FUNCTION_BLOCK FB_Security_System_Manager
  VAR_INPUT
    VI_System_Time_MS : UDINT;
    VI_IsActivePLC : BOOL;
    VI_Arm_Request : BOOL;
    VI_Disarm_Request : BOOL;
    VI_PIN_Code : STRING(4);
    VI_RFID_Tag : STRING(20);
    VI_2FA_Code : STRING(6);
    VI_Config : ST_Security_Global_Config;
    VI_Current_TOD : TOD;
  END_VAR
  VAR_OUTPUT
    VO_Armed : BOOL;
    VO_Alarm_Active : BOOL;
    VO_Siren_Active : BOOL;
    VO_Status_Msg : STRING(200);
    VO_Send_Code_Req : BOOL;
    VO_Code_To_Send : STRING(6);
  END_VAR
  VAR_IN_OUT
    VI_Motion_Sensors : ARRAY[1..16] OF BOOL;
    VI_Door_Sensors : ARRAY[1..GVL_CONSTANTS.C_MAX_DOOR_SENSORS] OF BOOL;
    VI_Window_Sensors : ARRAY[1..16] OF BOOL;
    VI_Bypass_Motion : ARRAY[1..16] OF BOOL;
    VI_Bypass_Doors : ARRAY[1..GVL_CONSTANTS.C_MAX_DOOR_SENSORS] OF BOOL;
    VI_Bypass_Windows : ARRAY[1..16] OF BOOL;
  END_VAR
  VAR
    L_i : INT;
    L_Any_Sensor_Active : BOOL;
    L_Arm_Delay_Timer : FB_System_Timer;
    L_Alarm_Delay_Timer : FB_System_Timer;
    L_Arming_In_Progress : BOOL;
    L_Valid_PIN : BOOL;
    fbAccessCode : FB_AccessCode_Manager;
    fbTwoFactor : FB_TwoFactor_Auth;
    L_2FA_Required : BOOL;
    L_Disarm_Pending : BOOL;
    L_Reset_2FA : BOOL;
    L_Auto_Arm_Trigger : BOOL;
    R_Trig_Auto_Arm : R_TRIG;
  END_VAR

            IF NOT VI_IsActivePLC THEN
    VO_Armed := FALSE;
    VO_Alarm_Active := FALSE;
    VO_Siren_Active := FALSE;
    VO_Send_Code_Req := FALSE;
    VO_Code_To_Send := '';
    VO_Status_Msg := 'Охрана: резервный ПЛК';
    L_Arming_In_Progress := FALSE;
    L_Disarm_Pending := FALSE;
    L_2FA_Required := FALSE;
    L_Reset_2FA := FALSE;
    RETURN;
END_IF;

// 1. Проверка PIN-кода или RFID-метки через менеджер кодов
fbAccessCode(
    VI_System_Time_MS := VI_System_Time_MS,
    VI_IsActivePLC := VI_IsActivePLC,
    VI_Code_To_Check := VI_PIN_Code,
    VI_RFID_To_Check := VI_RFID_Tag,
    VI_Access_Codes := GVL_RETAIN.G_Access_Codes,
    VI_RFID_Tags := GVL_RETAIN.G_RFID_Tags,
    VO_Code_Valid => L_Valid_PIN
);

// 2. Логика постановки на охрану (с задержкой на выход)
L_Auto_Arm_Trigger := FALSE;
IF VI_Config.auto_arm_enabled THEN
    IF VI_Current_TOD >= UDINT_TO_TOD(VI_Config.auto_arm_time_ms) THEN
        L_Auto_Arm_Trigger := TRUE;
    END_IF;
END_IF;
R_Trig_Auto_Arm(CLK := L_Auto_Arm_Trigger);

IF ((VI_Arm_Request AND L_Valid_PIN) OR R_Trig_Auto_Arm.Q) AND NOT VO_Armed AND NOT L_Arming_In_Progress THEN
    // Проверка, что все двери/окна закрыты перед постановкой (с учетом байпаса)
    L_Any_Sensor_Active := FALSE;
    FOR L_i := 1 TO GVL_CONSTANTS.C_MAX_DOOR_SENSORS DO IF VI_Door_Sensors[L_i] AND NOT VI_Bypass_Doors[L_i] THEN L_Any_Sensor_Active := TRUE; END_IF; END_FOR;
    FOR L_i := 1 TO 16 DO IF VI_Window_Sensors[L_i] AND NOT VI_Bypass_Windows[L_i] THEN L_Any_Sensor_Active := TRUE; END_IF; END_FOR;
    
    IF NOT L_Any_Sensor_Active THEN
        L_Arming_In_Progress := TRUE;
        VO_Status_Msg := 'Постановка на охрану. Покиньте помещение.';
    ELSE
        VO_Status_Msg := 'Ошибка постановки: Открыты двери или окна';
    END_IF;
END_IF;

L_Arm_Delay_Timer(IN := L_Arming_In_Progress, PT := TO_TIME(VI_Config.exit_delay_seconds * 1000), VI_System_Time_MS := VI_System_Time_MS);
IF L_Arm_Delay_Timer.Q THEN
    L_Arming_In_Progress := FALSE;
    VO_Armed := TRUE;
    VO_Status_Msg := 'Система под охраной';
END_IF;

// 3. Логика снятия с охраны с 2FA
IF VI_Disarm_Request AND L_Valid_PIN AND VO_Armed THEN
    IF VI_Config.enable_2fa THEN
        L_Disarm_Pending := TRUE;
        L_2FA_Required := TRUE;
        VO_Status_Msg := 'Ожидание 2FA для снятия с охраны';
    ELSE
        // Снятие без 2FA
        VO_Armed := FALSE;
        VO_Alarm_Active := FALSE;
        VO_Siren_Active := FALSE;
        L_Arming_In_Progress := FALSE;
        VO_Status_Msg := 'Система снята с охраны';
    END_IF;
END_IF;

fbTwoFactor(
    VI_System_Time_MS := VI_System_Time_MS,
    VI_Start_Auth := L_2FA_Required,
    VI_Method := E_TwoFactor_Method.TF_METHOD_TOTP, // Для примера
    VI_User_Code := VI_2FA_Code, // Используем отдельный вход для 2FA кода
    VI_Reset_Success := L_Reset_2FA
);

VO_Send_Code_Req := fbTwoFactor.VO_Send_Code_Req;
VO_Code_To_Send := fbTwoFactor.VO_Code_To_Send;

IF L_Disarm_Pending AND fbTwoFactor.VO_State.Is_Success THEN
    VO_Armed := FALSE;
    VO_Alarm_Active := FALSE;
    VO_Siren_Active := FALSE;
    L_Arming_In_Progress := FALSE;
    L_Disarm_Pending := FALSE;
    L_2FA_Required := FALSE;
    L_Reset_2FA := TRUE;
    VO_Status_Msg := 'Система снята с охраны';
ELSIF L_Disarm_Pending AND fbTwoFactor.VO_State.Is_Locked THEN
    L_Disarm_Pending := FALSE;
    L_2FA_Required := FALSE;
    L_Reset_2FA := FALSE;
    VO_Status_Msg := 'Ошибка 2FA: Превышено количество попыток';
ELSE
    L_Reset_2FA := FALSE;
END_IF;

// 4. Логика тревоги (с задержкой на вход)
IF VO_Armed THEN
    L_Any_Sensor_Active := FALSE;
    FOR L_i := 1 TO 16 DO IF VI_Motion_Sensors[L_i] AND NOT VI_Bypass_Motion[L_i] THEN L_Any_Sensor_Active := TRUE; END_IF; END_FOR;
    FOR L_i := 1 TO GVL_CONSTANTS.C_MAX_DOOR_SENSORS DO IF VI_Door_Sensors[L_i] AND NOT VI_Bypass_Doors[L_i] THEN L_Any_Sensor_Active := TRUE; END_IF; END_FOR;
    FOR L_i := 1 TO 16 DO IF VI_Window_Sensors[L_i] AND NOT VI_Bypass_Windows[L_i] THEN L_Any_Sensor_Active := TRUE; END_IF; END_FOR;
    
    // Защелкиваем факт нарушения периметра, чтобы кратковременное срабатывание датчика не сбрасывало таймер
    IF L_Any_Sensor_Active THEN
        L_Alarm_Delay_Timer.IN := TRUE;
    END_IF;
    
    L_Alarm_Delay_Timer(PT := TO_TIME(VI_Config.entry_delay_seconds * 1000), VI_System_Time_MS := VI_System_Time_MS);
    
    IF L_Alarm_Delay_Timer.Q THEN
        VO_Alarm_Active := TRUE;
        VO_Siren_Active := TRUE;
        VO_Status_Msg := 'ТРЕВОГА! Нарушение периметра';
    ELSIF L_Alarm_Delay_Timer.IN THEN
        VO_Status_Msg := 'Внимание! Введите PIN-код для отмены тревоги';
    END_IF;
ELSE
    L_Alarm_Delay_Timer(IN := FALSE, PT := T#0s, VI_System_Time_MS := VI_System_Time_MS); // Сброс таймера при снятии с охраны
END_IF;
// >>> BULK_SYNC_ANCHOR: FB_Security_System_Manager <<<
          
END_FUNCTION_BLOCK

FUNCTION_BLOCK FB_Heating_Runtime_Diagnostics_Phase
  VAR_INPUT
    VI_Enable : BOOL;
    VI_System_Time_MS : UDINT;
  END_VAR
  VAR_OUTPUT
    VO_Executed : BOOL;
    VO_Valid : BOOL;
  END_VAR
  VAR
    fbRootCauseDiagnostics : FB_Heating_RootCause_Diagnostics;
    fbDiagEventManager : FB_Diagnostics_Event_Manager;
    L_i : INT;
    L_Any_Heating_Device_OOS : BOOL;
    L_Critical_Fault : BOOL;
    L_Device_Text : STRING(200);
    L_Critical_Text : STRING(200);
    L_Event_Text : STRING(200);
    L_Add_Text : STRING(80);
  END_VAR

            // ==============================================================================
// Heating runtime diagnostics phase
// Owns diagnostics publication for heating runtime sequencing.
// Does NOT own heating control or output decisions.
// ==============================================================================



VO_Executed := FALSE;
VO_Valid := FALSE;

IF NOT VI_Enable THEN
    RETURN;
END_IF;

// ======================================================
// ROOT CAUSE DIAGNOSTICS
// ======================================================
fbRootCauseDiagnostics(
    VI_Enable := TRUE
);

// ======================================================
// DEFAULTS
// ======================================================
L_Any_Heating_Device_OOS := FALSE;
L_Critical_Fault := FALSE;
L_Device_Text := '';
L_Critical_Text := '';
L_Event_Text := '';
L_Add_Text := '';

// ======================================================
// SERVICE / OUT-OF-SERVICE FLAGS
// ======================================================
GVL_STATUS.G_Diagnostics.Backup_Pump_Out_Of_Service :=
    NOT GVL_CONFIG.G_Backup_Circulation_Pump_In_Service;

GVL_STATUS.G_Diagnostics.Electric_Heater_Out_Of_Service :=
    NOT GVL_CONFIG.G_Electric_Heater_In_Service;

IF GVL_STATUS.G_Diagnostics.Backup_Pump_Out_Of_Service THEN
    L_Any_Heating_Device_OOS := TRUE;
    L_Add_Text := 'backup pump out of service';
    L_Device_Text := L_Add_Text;
END_IF;

IF GVL_STATUS.G_Diagnostics.Electric_Heater_Out_Of_Service THEN
    L_Any_Heating_Device_OOS := TRUE;
    L_Add_Text := 'electric heater out of service';
    IF LEN(L_Device_Text) = 0 THEN
        L_Device_Text := L_Add_Text;
    ELSIF (LEN(L_Device_Text) + LEN(L_Add_Text) + 2) < 200 THEN
        L_Device_Text := CONCAT(L_Device_Text, CONCAT('; ', L_Add_Text));
    END_IF;
END_IF;

fbDiagEventManager(
    VI_Code := GVL_CONFIG.ERR_BACKUP_PUMP_OUT_OF_SERVICE,
    VI_Severity := 2,
    VI_Active := GVL_STATUS.G_Diagnostics.Backup_Pump_Out_Of_Service,
    VI_Timestamp := VI_System_Time_MS,
    VI_Source := 400,
    VIO_Events := GVL_STATUS.G_Diagnostics_Events,
    VIO_Count := GVL_STATUS.G_Diagnostics_Count
);

fbDiagEventManager(
    VI_Code := GVL_CONFIG.ERR_ELECTRIC_HEATER_OUT_OF_SERVICE,
    VI_Severity := 2,
    VI_Active := GVL_STATUS.G_Diagnostics.Electric_Heater_Out_Of_Service,
    VI_Timestamp := VI_System_Time_MS,
    VI_Source := 401,
    VIO_Events := GVL_STATUS.G_Diagnostics_Events,
    VIO_Count := GVL_STATUS.G_Diagnostics_Count
);

FOR L_i := 1 TO GVL_CONSTANTS.C_MAX_MANIFOLDS DO

    GVL_STATUS.G_Diagnostics.Manifold_Pump_Out_Of_Service[L_i] :=
        NOT GVL_CONFIG.G_Manifold_Pump_In_Service[L_i];

    IF GVL_STATUS.G_Diagnostics.Manifold_Pump_Out_Of_Service[L_i] THEN
        L_Any_Heating_Device_OOS := TRUE;
        L_Add_Text := CONCAT('manifold pump OOS #', INT_TO_STRING(L_i));

        IF LEN(L_Device_Text) = 0 THEN
            L_Device_Text := L_Add_Text;
        ELSIF (LEN(L_Device_Text) + LEN(L_Add_Text) + 2) < 200 THEN
            L_Device_Text := CONCAT(L_Device_Text, CONCAT('; ', L_Add_Text));
        END_IF;
    END_IF;

    fbDiagEventManager(
        VI_Code := GVL_CONFIG.ERR_MANIFOLD_PUMP_OUT_OF_SERVICE,
        VI_Severity := 2,
        VI_Active := GVL_STATUS.G_Diagnostics.Manifold_Pump_Out_Of_Service[L_i],
        VI_Timestamp := VI_System_Time_MS,
        VI_Source := 410 + L_i,
        VIO_Events := GVL_STATUS.G_Diagnostics_Events,
        VIO_Count := GVL_STATUS.G_Diagnostics_Count
    );

END_FOR;

GVL_STATUS.G_Diagnostics.DHW_Heating_Pump_Out_Of_Service :=
    NOT GVL_CONFIG.G_DHW_Heating_Pump_In_Service;

GVL_STATUS.G_Diagnostics.DHW_Circ_Pump_Out_Of_Service :=
    NOT GVL_CONFIG.G_DHW_Circ_Pump_In_Service;

IF GVL_STATUS.G_Diagnostics.DHW_Heating_Pump_Out_Of_Service THEN
    L_Any_Heating_Device_OOS := TRUE;
    L_Add_Text := 'DHW heating pump out of service';

    IF LEN(L_Device_Text) = 0 THEN
        L_Device_Text := L_Add_Text;
    ELSIF (LEN(L_Device_Text) + LEN(L_Add_Text) + 2) < 200 THEN
        L_Device_Text := CONCAT(L_Device_Text, CONCAT('; ', L_Add_Text));
    END_IF;
END_IF;

IF GVL_STATUS.G_Diagnostics.DHW_Circ_Pump_Out_Of_Service THEN
    L_Any_Heating_Device_OOS := TRUE;
    L_Add_Text := 'DHW circ pump out of service';

    IF LEN(L_Device_Text) = 0 THEN
        L_Device_Text := L_Add_Text;
    ELSIF (LEN(L_Device_Text) + LEN(L_Add_Text) + 2) < 200 THEN
        L_Device_Text := CONCAT(L_Device_Text, CONCAT('; ', L_Add_Text));
    END_IF;
END_IF;

fbDiagEventManager(
    VI_Code := GVL_CONFIG.ERR_DHW_HEATING_PUMP_OUT_OF_SERVICE,
    VI_Severity := 2,
    VI_Active := GVL_STATUS.G_Diagnostics.DHW_Heating_Pump_Out_Of_Service,
    VI_Timestamp := VI_System_Time_MS,
    VI_Source := 420,
    VIO_Events := GVL_STATUS.G_Diagnostics_Events,
    VIO_Count := GVL_STATUS.G_Diagnostics_Count
);

fbDiagEventManager(
    VI_Code := GVL_CONFIG.ERR_DHW_CIRC_PUMP_OUT_OF_SERVICE,
    VI_Severity := 2,
    VI_Active := GVL_STATUS.G_Diagnostics.DHW_Circ_Pump_Out_Of_Service,
    VI_Timestamp := VI_System_Time_MS,
    VI_Source := 421,
    VIO_Events := GVL_STATUS.G_Diagnostics_Events,
    VIO_Count := GVL_STATUS.G_Diagnostics_Count
);

// ======================================================
// FREEZE HARDWARE EVENT PROJECTION
// ======================================================
L_Critical_Fault := GVL_STATE.G_Freeze_Hardware_Failed;

IF L_Critical_Fault THEN
    L_Critical_Text := 'Freeze hardware critical fault';
END_IF;

fbDiagEventManager(
    VI_Code := GVL_CONFIG.ERR_FREEZE_HARDWARE_FAILED,
    VI_Severity := 4,
    VI_Active := L_Critical_Fault,
    VI_Timestamp := VI_System_Time_MS,
    VI_Source := 430,
    VIO_Events := GVL_STATUS.G_Diagnostics_Events,
    VIO_Count := GVL_STATUS.G_Diagnostics_Count
);

GVL_STATUS.G_Diagnostics.Freeze_Hardware_Event_Pending :=
    GVL_STATUS.G_Diagnostics.Freeze_Hardware_Event_Pending OR
    L_Critical_Fault OR
    L_Any_Heating_Device_OOS;

IF L_Critical_Fault AND L_Any_Heating_Device_OOS THEN
    L_Event_Text := CONCAT(L_Critical_Text, '; ');
    IF (LEN(L_Event_Text) + LEN(L_Device_Text)) < 200 THEN
        L_Event_Text := CONCAT(L_Event_Text, L_Device_Text);
    END_IF;
    GVL_STATUS.G_Diagnostics.Freeze_Hardware_Event_Text := L_Event_Text;
ELSIF L_Critical_Fault THEN
    GVL_STATUS.G_Diagnostics.Freeze_Hardware_Event_Text := L_Critical_Text;
ELSIF L_Any_Heating_Device_OOS THEN
    GVL_STATUS.G_Diagnostics.Freeze_Hardware_Event_Text := L_Device_Text;
END_IF;

VO_Executed := TRUE;
VO_Valid := TRUE;

// >>> BULK_SYNC_ANCHOR: FB_Heating_Runtime_Diagnostics_Phase <<<
          
END_FUNCTION_BLOCK

FUNCTION_BLOCK FB_Heating_Thermal_Model
  VAR
    L_i : INT;
    L_DeltaT : REAL;
    L_Loss : REAL;
    L_Gain : REAL;
    L_Outdoor : REAL;
  END_VAR

            L_Outdoor := GVL_STATE.G_Outdoor_Temp;

FOR L_i := 1 TO GVL_CONSTANTS.C_MAX_ZONES DO

    L_DeltaT := GVL_STATE.G_Room_Temps[L_i] - L_Outdoor;

    L_Loss := L_DeltaT * REAL#0.01 * GVL_HEATING_POLICY.G_Zone_Thermal_Inertia[L_i];

    L_Gain := (GVL_STATE.G_Floor_Temps[L_i] - GVL_STATE.G_Room_Temps[L_i]) * REAL#0.05;

    GVL_HEATING_POLICY.G_Zone_Heat_Loss_Rate[L_i] := L_Loss;
    GVL_HEATING_POLICY.G_Zone_Heat_Gain_Rate[L_i] := L_Gain;

    GVL_HEATING_POLICY.G_Zone_Thermal_Response[L_i] := L_Gain - L_Loss;

    GVL_HEATING_POLICY.G_Zone_Thermal_Demand[L_i] := 
        GVL_STATE.G_Target_Temperature - GVL_STATE.G_Room_Temps[L_i];

    IF ABS(GVL_HEATING_POLICY.G_Zone_Thermal_Response[L_i]) > REAL#0.01 THEN
        GVL_HEATING_POLICY.G_Zone_Time_To_Heat_MS[L_i] := 
            REAL_TO_UDINT(ABS(GVL_HEATING_POLICY.G_Zone_Thermal_Demand[L_i] /
                  GVL_HEATING_POLICY.G_Zone_Thermal_Response[L_i]) * REAL#60000.0);
    ELSE
        GVL_HEATING_POLICY.G_Zone_Time_To_Heat_MS[L_i] := 0;
    END_IF;

    GVL_HEATING_POLICY.G_Zone_Predicted_Temp_30m[L_i] :=
        GVL_STATE.G_Room_Temps[L_i] + 
        GVL_HEATING_POLICY.G_Zone_Thermal_Response[L_i] * REAL#30.0;

    GVL_HEATING_POLICY.G_Zone_Thermal_Model_Confidence[L_i] :=
        LIMIT(REAL#0.0, REAL#1.0, ABS(GVL_HEATING_POLICY.G_Zone_Thermal_Response[L_i]));

END_FOR;
          
END_FUNCTION_BLOCK

FUNCTION_BLOCK FB_Gateway_Interface
  VAR_INPUT
    VI_System_Time_MS : UDINT;
    VI_Local_PLC_Role : E_PLC_ROLE;
    VI_Incoming_Command : ST_Gateway_Command;
    VI_Command_Received : BOOL;
    VI_Outdoor_Temp : REAL;
    VI_Security_Armed : BOOL;
    VI_Flood_Alarm_Active : BOOL;
    VI_Gas_Alarm_Active : BOOL;
    VI_Fire_Alarm_Active : BOOL;
    VI_Methane_Concentration : REAL;
    VI_Active_Scenario : E_SCENARIO_TYPE;
    VI_Send_2FA_Req : BOOL;
    VI_2FA_Code : STRING(6);
  END_VAR
  VAR_OUTPUT
    VO_Modbus_Registers : ARRAY[0..GVL_CONSTANTS.C_MAX_MODBUS_REGISTERS-1] OF WORD;
    VO_Lighting_Override : ARRAY[1..GVL_CONSTANTS.C_MAX_LIGHT_ZONES] OF BYTE;
    VO_Blinds_Override : ARRAY[1..GVL_CONSTANTS.C_MAX_BLINDS] OF BYTE;
    VO_Socket_Override : ARRAY[1..GVL_CONSTANTS.C_MAX_SOCKETS] OF BOOL;
    VO_Arm_Req : BOOL;
    VO_Disarm_Req : BOOL;
    VO_PIN_Code : STRING(4);
    VO_RFID_Tag : STRING(20);
    VO_2FA_Code_In : STRING(6);
    VO_Data_Ready : BOOL;
    VO_HMI_Status_Message : STRING(200);
    VO_Telegram_Msg : STRING(200);
    VO_Send_Telegram : BOOL;
    VO_Set_Scenario_Req : BOOL;
    VO_Target_Scenario : E_SCENARIO_TYPE;
    VO_Set_Temp_Req : BOOL;
    VO_Target_Zone : INT;
    VO_Target_Temp : REAL;
    VO_Set_Vent_Req : BOOL;
    VO_Target_Vent_Speed : BYTE;
    VO_Reset_Errors_Req : BOOL;
    VO_Set_Config_Req : BOOL;
    VO_Sync_Time_Req : BOOL;
    VO_New_Time_MS : UDINT;
  END_VAR
  VAR_IN_OUT
    VI_FloorHeating_Temps : ARRAY[1..GVL_CONSTANTS.C_MAX_HEATING_CIRCUITS] OF REAL;
    VI_Room_Temps : ARRAY[1..GVL_CONSTANTS.C_MAX_ZONES] OF REAL;
    VI_Zone_Valve_States : ARRAY[1..GVL_CONSTANTS.C_MAX_HEATING_CIRCUITS] OF BOOL;
    VI_Manifold_Pressures : ARRAY[1..GVL_CONSTANTS.C_MAX_MANIFOLDS] OF REAL;
    VI_Manifold_Pump_States : ARRAY[1..GVL_CONSTANTS.C_MAX_MANIFOLDS] OF BOOL;
    VI_Lighting_Base_Levels : ARRAY[1..GVL_CONSTANTS.C_MAX_LIGHT_ZONES] OF BYTE;
    VI_Socket_States : ARRAY[1..GVL_CONSTANTS.C_MAX_SOCKETS] OF BOOL;
    VI_Blinds_Positions : ARRAY[1..GVL_CONSTANTS.C_MAX_BLINDS] OF BYTE;
    VI_Allowed_IPs : ARRAY[1..GVL_CONSTANTS.C_MAX_ALLOWED_IPS] OF STRING(15);
  END_VAR
  VAR
    L_last_update_time : UDINT;
    L_i : INT;
    L_j : INT;
    L_idx : INT;
    L_tmp_word : WORD;
    L_Code_UDINT : UDINT;
    L_Prev_Fire : BOOL;
    L_Prev_Gas : BOOL;
    L_Prev_Flood : BOOL;
    L_Prev_Security : BOOL;
    L_Deduplicator : FB_Command_Deduplication;
    L_CRC_Calc : FB_CRC32_Calculator;
    L_Calculated_CRC : DWORD;
    L_IP_Allowed : BOOL;
    L_Process_Command : ST_Gateway_Command;
    L_Has_Command_To_Process : BOOL;
  END_VAR
  VAR RETAIN
    L_Command_Buffer : ARRAY[1..GVL_CONSTANTS.C_MAX_GATEWAY_COMMANDS] OF ST_Gateway_Command;
    L_Buffer_Head : INT := 1;
    L_Buffer_Tail : INT := 1;
    L_Buffer_Count : INT := 0;
  END_VAR

            VO_Send_Telegram := FALSE;
IF VI_Fire_Alarm_Active AND NOT L_Prev_Fire THEN
    VO_Telegram_Msg := 'ВНИМАНИЕ! ПОЖАРНАЯ ТРЕВОГА!';
    VO_Send_Telegram := TRUE;
END_IF;
IF VI_Gas_Alarm_Active AND NOT L_Prev_Gas THEN
    VO_Telegram_Msg := 'ВНИМАНИЕ! УТЕЧКА ГАЗА!';
    VO_Send_Telegram := TRUE;
END_IF;
IF VI_Flood_Alarm_Active AND NOT L_Prev_Flood THEN
    VO_Telegram_Msg := 'ВНИМАНИЕ! ПРОТЕЧКА ВОДЫ!';
    VO_Send_Telegram := TRUE;
END_IF;
IF VI_Security_Armed AND NOT L_Prev_Security THEN
    VO_Telegram_Msg := 'ОХРАНА ВКЛЮЧЕНА';
    VO_Send_Telegram := TRUE;
ELSIF NOT VI_Security_Armed AND L_Prev_Security THEN
    VO_Telegram_Msg := 'ОХРАНА ОТКЛЮЧЕНА';
    VO_Send_Telegram := TRUE;
END_IF;

L_Prev_Fire := VI_Fire_Alarm_Active;
L_Prev_Gas := VI_Gas_Alarm_Active;
L_Prev_Flood := VI_Flood_Alarm_Active;
L_Prev_Security := VI_Security_Armed;

IF (VI_System_Time_MS - L_last_update_time) >= GVL_CONSTANTS.C_MS_IN_SECOND THEN
    L_last_update_time := VI_System_Time_MS;
    L_tmp_word := 0;
    IF VI_Local_PLC_Role = E_PLC_ROLE.ROLE_ACTIVE THEN L_tmp_word := L_tmp_word OR 1; END_IF;
    IF VI_Security_Armed THEN L_tmp_word := L_tmp_word OR 2; END_IF;
    IF VI_Flood_Alarm_Active THEN L_tmp_word := L_tmp_word OR 4; END_IF;
    IF VI_Gas_Alarm_Active THEN L_tmp_word := L_tmp_word OR 8; END_IF;
    IF VI_Fire_Alarm_Active THEN L_tmp_word := L_tmp_word OR 16; END_IF;
    VO_Modbus_Registers[0] := L_tmp_word;

    FOR L_i := 1 TO GVL_CONSTANTS.C_MAX_HEATING_CIRCUITS DO
        VO_Modbus_Registers[L_i] := TO_WORD(TO_INT(VI_FloorHeating_Temps[L_i] * REAL#10.0));
    END_FOR;

    FOR L_i := 1 TO GVL_CONSTANTS.C_MAX_ZONES DO
        VO_Modbus_Registers[16 + L_i] := TO_WORD(TO_INT(VI_Room_Temps[L_i] * REAL#10.0));
    END_FOR;

    L_tmp_word := 0;
    FOR L_i := 1 TO GVL_CONSTANTS.C_MAX_HEATING_CIRCUITS DO
        IF VI_Zone_Valve_States[L_i] THEN
            L_tmp_word := L_tmp_word OR SHL(TO_WORD(1), L_i - 1);
        END_IF;
    END_FOR;
    VO_Modbus_Registers[33] := L_tmp_word;

    FOR L_i := 1 TO GVL_CONSTANTS.C_MAX_MANIFOLDS DO
        VO_Modbus_Registers[33 + L_i] := TO_WORD(TO_INT(VI_Manifold_Pressures[L_i] * REAL#100.0));
    END_FOR;

    FOR L_i := 1 TO GVL_CONSTANTS.C_MAX_LIGHT_ZONES DO
        VO_Modbus_Registers[39 + L_i] := TO_WORD(VI_Lighting_Base_Levels[L_i]);
    END_FOR;

    FOR L_i := 1 TO GVL_CONSTANTS.C_MAX_BLINDS DO
        VO_Modbus_Registers[71 + L_i] := TO_WORD(VI_Blinds_Positions[L_i]);
    END_FOR;

    FOR L_i := 0 TO (GVL_CONSTANTS.C_MAX_SOCKETS - 1) / 16 DO
        L_tmp_word := 0;
        FOR L_j := 1 TO 16 DO
            L_idx := (L_i * 16) + L_j;
            IF L_idx <= GVL_CONSTANTS.C_MAX_SOCKETS THEN
                IF VI_Socket_States[L_idx] THEN
                    L_tmp_word := L_tmp_word OR SHL(TO_WORD(1), L_j - 1);
                END_IF;
            END_IF;
        END_FOR;
        VO_Modbus_Registers[92 + L_i] := L_tmp_word;
    END_FOR;

    VO_Modbus_Registers[100] := SEL(VI_Send_2FA_Req, 0, 1);
    IF VI_Send_2FA_Req THEN
        L_Code_UDINT := STRING_TO_UDINT(VI_2FA_Code);
        VO_Modbus_Registers[101] := TO_WORD(L_Code_UDINT AND 16#FFFF);
        VO_Modbus_Registers[102] := TO_WORD(SHR(L_Code_UDINT, 16));
    ELSE
        VO_Modbus_Registers[101] := 0;
        VO_Modbus_Registers[102] := 0;
    END_IF;

    VO_Data_Ready := TRUE;
END_IF;

VO_Arm_Req := FALSE;
VO_Disarm_Req := FALSE;
VO_Set_Scenario_Req := FALSE;
VO_Set_Temp_Req := FALSE;
VO_Set_Vent_Req := FALSE;
VO_Reset_Errors_Req := FALSE;
VO_Set_Config_Req := FALSE;
VO_Sync_Time_Req := FALSE;
L_Has_Command_To_Process := FALSE;

IF VI_Command_Received THEN
    IF VI_Local_PLC_Role = E_PLC_ROLE.ROLE_ACTIVE THEN
        L_Process_Command := VI_Incoming_Command;
        L_Has_Command_To_Process := TRUE;
    ELSE
        IF L_Buffer_Count < GVL_CONSTANTS.C_MAX_GATEWAY_COMMANDS THEN
            L_Command_Buffer[L_Buffer_Head] := VI_Incoming_Command;
            L_Buffer_Head := L_Buffer_Head + 1;
            IF L_Buffer_Head > GVL_CONSTANTS.C_MAX_GATEWAY_COMMANDS THEN L_Buffer_Head := 1; END_IF;
            L_Buffer_Count := L_Buffer_Count + 1;
        END_IF;
    END_IF;
END_IF;

IF NOT L_Has_Command_To_Process AND (VI_Local_PLC_Role = E_PLC_ROLE.ROLE_ACTIVE) AND (L_Buffer_Count > 0) THEN
    L_Process_Command := L_Command_Buffer[L_Buffer_Tail];
    L_Buffer_Tail := L_Buffer_Tail + 1;
    IF L_Buffer_Tail > GVL_CONSTANTS.C_MAX_GATEWAY_COMMANDS THEN L_Buffer_Tail := 1; END_IF;
    L_Buffer_Count := L_Buffer_Count - 1;
    L_Has_Command_To_Process := TRUE;
END_IF;

IF L_Has_Command_To_Process THEN
    L_IP_Allowed := FALSE;
    IF L_Process_Command.source_ip = '' THEN
        L_IP_Allowed := TRUE;
    ELSE
        FOR L_i := 1 TO GVL_CONSTANTS.C_MAX_ALLOWED_IPS DO
            IF VI_Allowed_IPs[L_i] = L_Process_Command.source_ip THEN
                L_IP_Allowed := TRUE;
                EXIT;
            END_IF;
        END_FOR;
    END_IF;

    IF NOT L_IP_Allowed THEN
        VO_HMI_Status_Message := 'Gateway: Ошибка безопасности (Неизвестный IP)';
        RETURN;
    END_IF;

    L_CRC_Calc();
    L_Calculated_CRC := L_CRC_Calc.VO_CRC;

    IF L_Calculated_CRC = L_Process_Command.crc32 THEN
        L_Deduplicator(VI_Command_ID := L_Process_Command.command_id, VI_Command_Type := L_Process_Command.command_type, VI_Command_Value := L_Process_Command.target_value, VI_System_Time_MS := VI_System_Time_MS);

        IF L_Deduplicator.VO_Is_New_Command THEN
            CASE L_Process_Command.command_type OF
                E_Gateway_Command_Type.CMD_SET_SCENARIO:
                    VO_Set_Scenario_Req := TRUE;
                    VO_Target_Scenario := L_Process_Command.target_scenario;
                    VO_HMI_Status_Message := 'Gateway: Сценарий изменен';
                E_Gateway_Command_Type.CMD_SET_LIGHT:
                    IF (L_Process_Command.target_zone >= 1) AND (L_Process_Command.target_zone <= GVL_CONSTANTS.C_MAX_LIGHT_ZONES) THEN
                        VO_Lighting_Override[L_Process_Command.target_zone] := TO_BYTE(L_Process_Command.target_value);
                        VO_HMI_Status_Message := 'Gateway: Команда освещения принята';
                    END_IF;
                E_Gateway_Command_Type.CMD_SET_BLINDS:
                    IF (L_Process_Command.target_zone >= 1) AND (L_Process_Command.target_zone <= GVL_CONSTANTS.C_MAX_BLINDS) THEN
                        VO_Blinds_Override[L_Process_Command.target_zone] := TO_BYTE(L_Process_Command.target_value);
                        VO_HMI_Status_Message := 'Gateway: Команда штор принята';
                    END_IF;
                E_Gateway_Command_Type.CMD_SET_SOCKET:
                    IF (L_Process_Command.target_zone >= 1) AND (L_Process_Command.target_zone <= GVL_CONSTANTS.C_MAX_SOCKETS) THEN
                        VO_Socket_Override[L_Process_Command.target_zone] := L_Process_Command.target_on_off;
                        VO_HMI_Status_Message := 'Gateway: Команда розетки принята';
                    END_IF;
                E_Gateway_Command_Type.CMD_SET_SECURITY:
                    IF L_Process_Command.target_armed THEN VO_Arm_Req := TRUE; ELSE VO_Disarm_Req := TRUE; END_IF;
                    VO_PIN_Code := L_Process_Command.target_pin;
                    VO_2FA_Code_In := L_Process_Command.target_2fa_code;
                    VO_HMI_Status_Message := 'Gateway: Запрос охраны принят';
                E_Gateway_Command_Type.CMD_SET_TEMP:
                    IF (L_Process_Command.target_zone >= 1) AND (L_Process_Command.target_zone <= GVL_CONSTANTS.C_MAX_HEATING_CIRCUITS) THEN
                        VO_Set_Temp_Req := TRUE;
                        VO_Target_Zone := L_Process_Command.target_zone;
                        VO_Target_Temp := L_Process_Command.target_value;
                        VO_HMI_Status_Message := 'Gateway: Уставка температуры изменена';
                    END_IF;
                E_Gateway_Command_Type.CMD_SET_VENT:
                    VO_Set_Vent_Req := TRUE;
                    VO_Target_Vent_Speed := TO_BYTE(L_Process_Command.target_value);
                    VO_HMI_Status_Message := 'Gateway: Уставка вентиляции изменена';
                E_Gateway_Command_Type.CMD_TELEGRAM_MSG:
                    VO_Telegram_Msg := L_Process_Command.telegram_msg;
                    VO_Send_Telegram := TRUE;
                    VO_HMI_Status_Message := 'Gateway: Сообщение Telegram отправлено';
                E_Gateway_Command_Type.CMD_SYNC_TIME:
                    VO_Sync_Time_Req := TRUE;
                    VO_New_Time_MS := REAL_TO_UDINT(L_Process_Command.target_value);
                    VO_HMI_Status_Message := 'Gateway: Время синхронизировано';
                E_Gateway_Command_Type.CMD_RESET_ERRORS:
                    VO_Reset_Errors_Req := TRUE;
                    VO_HMI_Status_Message := 'Gateway: Запрос на сброс ошибок принят';
                E_Gateway_Command_Type.CMD_SET_CONFIG:
                    VO_Set_Config_Req := TRUE;
                    VO_HMI_Status_Message := 'Gateway: Запрос на применение конфигурации принят';
            END_CASE;
        END_IF;
    ELSE
        VO_HMI_Status_Message := 'Gateway: Ошибка CRC команды';
    END_IF;
END_IF;

// >>> BULK_SYNC_ANCHOR: FB_Gateway_Interface <<<
          
END_FUNCTION_BLOCK

FUNCTION_BLOCK FB_Heating_Manifold_Control
  VAR_INPUT
    VI_System_Time_MS : UDINT;
    VI_IsActivePLC : BOOL;
    VI_DHW_Heating_Demand : BOOL;
    VI_Freeze_Mode_Active : BOOL;
    VI_Target_Supply_Temp : REAL;
    VI_Any_Zone_Active : ARRAY[1..GVL_CONSTANTS.C_MAX_MANIFOLDS] OF BOOL;
  END_VAR
  VAR_OUTPUT
    VO_Manifold_Pumps : ARRAY[1..GVL_CONSTANTS.C_MAX_MANIFOLDS] OF BOOL;
    VO_Manifold_Valves : ARRAY[1..GVL_CONSTANTS.C_MAX_MANIFOLDS] OF REAL;
    VO_Status : ARRAY[1..GVL_CONSTANTS.C_MAX_MANIFOLDS] OF ST_Manifold_Status;
  END_VAR
  VAR_IN_OUT
    VI_Manifold_Pressures : ARRAY[1..GVL_CONSTANTS.C_MAX_MANIFOLDS] OF REAL;
    VI_Manifold_Currents : ARRAY[1..GVL_CONSTANTS.C_MAX_MANIFOLDS] OF REAL;
    VI_Manifold_Temps_Supply : ARRAY[1..GVL_CONSTANTS.C_MAX_MANIFOLDS] OF REAL;
    VI_Manifold_Temps_Return : ARRAY[1..GVL_CONSTANTS.C_MAX_MANIFOLDS] OF REAL;
  END_VAR
  VAR
    L_i : INT;
    L_Delta_T : REAL;
    L_PID_Valves : ARRAY[1..GVL_CONSTANTS.C_MAX_MANIFOLDS] OF FB_PID_Controller;
    L_PID_Timer : ARRAY[1..GVL_CONSTANTS.C_MAX_MANIFOLDS] OF FB_System_Timer;
    L_Pump_Run_Timer : ARRAY[1..GVL_CONSTANTS.C_MAX_MANIFOLDS] OF FB_System_Timer;
    L_Pump_Pause_Timer : ARRAY[1..GVL_CONSTANTS.C_MAX_MANIFOLDS] OF FB_System_Timer;
    L_Pump_In_Pause : ARRAY[1..GVL_CONSTANTS.C_MAX_MANIFOLDS] OF BOOL;
    L_Pump_Diag : ARRAY[1..GVL_CONSTANTS.C_MAX_MANIFOLDS] OF FB_Device_Predictive_Diag;
  END_VAR

            // ==============================================================================
// Heating manifold control helper
// Internal refactoring helper for FB_Heating_System_Manager.
// Valve test override remains in FB_Heating_System_Manager for now.
// ==============================================================================



FOR L_i := 1 TO GVL_CONSTANTS.C_MAX_MANIFOLDS DO
    L_PID_Timer[L_i](IN := TRUE, PT := T#1s, VI_System_Time_MS := VI_System_Time_MS);
    IF L_PID_Timer[L_i].Q THEN
        L_PID_Timer[L_i](IN := FALSE, PT := T#1s, VI_System_Time_MS := VI_System_Time_MS);
        L_PID_Timer[L_i](IN := TRUE, PT := T#1s, VI_System_Time_MS := VI_System_Time_MS);

        L_PID_Valves[L_i](
            VI_SetPoint := VI_Target_Supply_Temp,
            VI_ProcessValue := VI_Manifold_Temps_Supply[L_i],
            VI_Kp := 2.0,
            VI_Tn := 120.0,
            VI_Tv := 0.0,
            VI_Y_Min := 0.0,
            VI_Y_Max := 100.0,
            VI_Cycle_Time_S := 1.0,
            VO_Output => VO_Manifold_Valves[L_i]
        );
    END_IF;

    L_Pump_Run_Timer[L_i](
        IN := VO_Manifold_Pumps[L_i] AND NOT L_Pump_In_Pause[L_i],
        PT := T#72h,
        VI_System_Time_MS := VI_System_Time_MS
    );
    IF L_Pump_Run_Timer[L_i].Q THEN
        L_Pump_In_Pause[L_i] := TRUE;
    END_IF;

    L_Pump_Pause_Timer[L_i](
        IN := L_Pump_In_Pause[L_i],
        PT := T#1h,
        VI_System_Time_MS := VI_System_Time_MS
    );
    IF L_Pump_Pause_Timer[L_i].Q THEN
        L_Pump_In_Pause[L_i] := FALSE;
    END_IF;

    IF VI_DHW_Heating_Demand THEN
        VO_Manifold_Pumps[L_i] := FALSE;
        VO_Manifold_Valves[L_i] := 0.0;
    ELSE
        VO_Manifold_Pumps[L_i] := VI_IsActivePLC AND VI_Any_Zone_Active[L_i] AND NOT L_Pump_In_Pause[L_i];
    END_IF;

    IF VI_Freeze_Mode_Active THEN
        VO_Manifold_Pumps[L_i] := TRUE;
        IF VO_Manifold_Valves[L_i] < 35.0 THEN
            VO_Manifold_Valves[L_i] := 35.0;
        END_IF;
    END_IF;

    VO_Status[L_i].Pump_On := VO_Manifold_Pumps[L_i];
    VO_Status[L_i].Pump_Current := VI_Manifold_Currents[L_i];
    VO_Status[L_i].Pressure := VI_Manifold_Pressures[L_i];
    VO_Status[L_i].Temp_Supply := VI_Manifold_Temps_Supply[L_i];
    VO_Status[L_i].Temp_Return := VI_Manifold_Temps_Return[L_i];
    VO_Status[L_i].Valve_Pos := VO_Manifold_Valves[L_i];

    L_Pump_Diag[L_i](
        VI_Current_Value := VI_Manifold_Currents[L_i],
        VI_Nominal_Value := 0.55,
        VI_Is_Running := VO_Manifold_Pumps[L_i],
        VI_Reset_Stats := FALSE,
        VI_System_Time_MS := VI_System_Time_MS,
        VIO_Health_Data := VO_Status[L_i].Health
    );

    IF VO_Manifold_Pumps[L_i] THEN
        L_Delta_T := VI_Manifold_Temps_Supply[L_i] - VI_Manifold_Temps_Return[L_i];

        VO_Status[L_i].Error := FALSE;
        VO_Status[L_i].Error_ID := 0;

        IF VI_Manifold_Currents[L_i] <= 0.01 THEN
            VO_Status[L_i].Error := TRUE;
            VO_Status[L_i].Error_ID := TO_WORD(GVL_CONFIG.ERR_PUMP_NO_CURRENT);
        ELSIF VI_Manifold_Currents[L_i] < 0.3 THEN
            VO_Status[L_i].Error := TRUE;
            VO_Status[L_i].Error_ID := TO_WORD(GVL_CONFIG.ERR_PUMP_UNDERCURRENT);
        ELSIF VI_Manifold_Currents[L_i] > 1.5 THEN
            VO_Status[L_i].Error := TRUE;
            VO_Status[L_i].Error_ID := TO_WORD(GVL_CONFIG.ERR_PUMP_OVERCURRENT);
        END_IF;

        IF (NOT VO_Status[L_i].Error) AND ((VI_Manifold_Pressures[L_i] < 1.5) OR (VI_Manifold_Pressures[L_i] > 2.5)) THEN
            VO_Status[L_i].Error := TRUE;
            VO_Status[L_i].Error_ID := TO_WORD(GVL_CONFIG.ERR_PRESSURE_OUT_OF_RANGE);
        END_IF;

        IF NOT VO_Status[L_i].Error THEN
            IF L_Delta_T < 5.0 THEN
                VO_Status[L_i].Error := TRUE;
                VO_Status[L_i].Error_ID := TO_WORD(GVL_CONFIG.ERR_DELTA_T_LOW);
            ELSIF L_Delta_T > 10.0 THEN
                VO_Status[L_i].Error := TRUE;
                VO_Status[L_i].Error_ID := TO_WORD(GVL_CONFIG.ERR_DELTA_T_HIGH);
            END_IF;
        END_IF;
    END_IF;
END_FOR;

// >>> BULK_SYNC_ANCHOR: FB_Heating_Manifold_Control <<<
          
END_FUNCTION_BLOCK

FUNCTION_BLOCK FB_Distributed_Orchestration_Runtime
  VAR_INPUT
    VI_Enable : BOOL;
    VI_System_Time_MS : UDINT;
  END_VAR
  VAR
    L_State : ST_Distributed_Orchestration_State;
    L_Finalized_Runtime_Continuity : BOOL;
  END_VAR

            IF NOT VI_Enable THEN
    GVL_Distributed_Orchestration.G_Runtime_Valid := FALSE;
    RETURN;
END_IF;

L_State.Runtime_Valid := TRUE;
L_State.Runtime_System_Time_MS := VI_System_Time_MS;

L_State.Orchestration_Sequence_Id :=
    GVL_Distributed_Orchestration.G_Last_Distributed_Sequence_Id + 1;

L_State.Distributed_Execution_Active := TRUE;

L_State.Cross_Node_Isolation_Required :=
    GVL_Distributed_Orchestration.G_Cross_Node_Isolation_Active;

L_State.Cross_Node_Recovery_Required :=
    GVL_Distributed_Orchestration.G_Cross_Node_Recovery_Active;

L_State.Cross_Node_Rollback_Required :=
    GVL_Distributed_Orchestration.G_Cross_Node_Rollback_Active;

L_Finalized_Runtime_Continuity :=
    GVL_SEMANTIC_PROGRESS.Semantic_Forward_Progress_Valid
    AND GVL_SEMANTIC_PROGRESS.Semantic_Execution_Continuity_OK
    AND NOT GVL_SEMANTIC_PROGRESS.Semantic_Progress_Lease_Expired
    AND NOT GVL_SEMANTIC_PROGRESS.Semantic_Progress_Quarantine_Active
    AND GVL_RUNTIME_SNAPSHOT.Snapshot_Frozen
    AND GVL_RUNTIME_SNAPSHOT.Snapshot_Publication_Allowed
    AND GVL_RUNTIME_SNAPSHOT.Snapshot_Copy_Valid
    AND GVL_RUNTIME_SNAPSHOT.Snapshot_Isolation_Valid
    AND NOT GVL_RUNTIME_SNAPSHOT.Snapshot_Mutation_Detected
    AND GVL_DISTRIBUTED_SNAPSHOT.Distributed_Publication_Reconciled
    AND GVL_DISTRIBUTED_SNAPSHOT.Distributed_Publication_Freeze_Valid
    AND GVL_DISTRIBUTED_SNAPSHOT.Distributed_Snapshot_Consistent
    AND GVL_DISTRIBUTED_COMMIT.Distributed_Commit_Valid
    AND GVL_DISTRIBUTED_COMMIT.Publication_Prepare_Valid
    AND GVL_DISTRIBUTED_COMMIT.Publication_Commit_Confirmed
    AND NOT GVL_DISTRIBUTED_COMMIT.Peer_Commit_Mismatch
    AND NOT GVL_DISTRIBUTED_COMMIT.Commit_Lease_Expired
    AND GVL_OUTPUT_EPOCH.Output_Publication_Valid
    AND GVL_OUTPUT_EPOCH.Output_Runtime_Epoch_Valid
    AND NOT GVL_OUTPUT_EPOCH.Output_Lease_Expired
    AND NOT GVL_OUTPUT_EPOCH.Output_Forced_Safe_Decay
    AND GVL_COMMAND_VERIFY.PreOutput_Barrier_OK
    AND NOT GVL_COMMAND_VERIFY.PreOutput_Block_IO;

L_State.Distributed_Scheduler_Healthy :=
    GVL_Runtime_Bus.G_TX_Healthy
    AND GVL_Distributed_Runtime.G_Distributed_Authority_Healthy
    AND L_Finalized_Runtime_Continuity;

L_State.Distributed_Timing_Window_Valid :=
    GVL_Distributed_Authority.G_Distributed_Safety_Barrier_OK
    AND L_Finalized_Runtime_Continuity;

IF L_State.Distributed_Scheduler_Healthy
   AND L_State.Distributed_Timing_Window_Valid THEN
    L_State.Distributed_Projection_Granted := TRUE;
    L_State.Distributed_Recovery_Allowed := TRUE;
    L_State.Distributed_Rollback_Allowed := TRUE;
    L_State.Status_Code := 0;
    L_State.Status_Text := 'Distributed orchestration runtime healthy';
ELSE
    L_State.Distributed_Projection_Blocked := TRUE;
    L_State.Distributed_Conflict_Detected := TRUE;
    L_State.Status_Code := 2;
    L_State.Status_Text := 'Distributed orchestration blocked';
END_IF;

IF GVL_Distributed_Runtime.G_Split_Brain_Suspected THEN
    L_State.Distributed_Split_Execution_Suspected := TRUE;
    L_State.Distributed_Projection_Blocked := TRUE;
    L_State.Status_Code := 3;
    L_State.Status_Text := 'Distributed split execution suspected';
END_IF;

GVL_Distributed_Orchestration.G_Orchestration_State := L_State;
GVL_Distributed_Orchestration.G_Last_Distributed_Sequence_Id := L_State.Orchestration_Sequence_Id;
GVL_Distributed_Orchestration.G_Distributed_Projection_Healthy := L_State.Distributed_Projection_Granted;
GVL_Distributed_Orchestration.G_Distributed_Scheduler_Healthy := L_State.Distributed_Scheduler_Healthy;
GVL_Distributed_Orchestration.G_Runtime_Valid := TRUE;
GVL_Distributed_Orchestration.G_Last_Update_MS := VI_System_Time_MS;
GVL_Distributed_Orchestration.G_Status_Code := L_State.Status_Code;
GVL_Distributed_Orchestration.G_Status_Text := L_State.Status_Text;
          
END_FUNCTION_BLOCK

FUNCTION_BLOCK FB_Boiler_Cascade_Manager
  VAR_INPUT
    VI_Enable : BOOL;
    VI_System_Time_MS : UDINT;
    VI_Boiler_Stop : BOOL;
    VI_DHW_Heating_Demand : BOOL;
    VI_DHW_Target_Temp : REAL;
    VI_Target_Supply_Temp : REAL;
    VI_Demand_Power : REAL;
    VI_Boiler_Flame_Status : ARRAY[1..GVL_CONSTANTS.C_MAX_BOILERS] OF BOOL;
    VI_Boiler_Error_Status : ARRAY[1..GVL_CONSTANTS.C_MAX_BOILERS] OF BOOL;
    VI_Boiler_OT_Online : ARRAY[1..GVL_CONSTANTS.C_MAX_BOILERS] OF BOOL;
    VI_Boiler_Modulation : ARRAY[1..GVL_CONSTANTS.C_MAX_BOILERS] OF REAL;
  END_VAR
  VAR_OUTPUT
    VO_Boiler_Enable : ARRAY[1..GVL_CONSTANTS.C_MAX_BOILERS] OF BOOL;
    VO_Boiler_Setpoint : ARRAY[1..GVL_CONSTANTS.C_MAX_BOILERS] OF REAL;
    VO_Lead_Boiler : BYTE;
  END_VAR
  VAR
    L_i : INT;
    L_Lead_Boiler : BYTE := 1;
    L_Last_Rotation_MS : UDINT := 0;
    L_Rotation_Initialized : BOOL := FALSE;
    L_Rotation_Period_MS : UDINT := 604800000;
    L_Lead_Available : BOOL;
    L_Reserve_Available : BOOL;
    L_Reserve_Boiler : BYTE;
    L_Start_Reserve : BOOL;
    L_Target_Setpoint : REAL;
    L_Flame_Miss_Timer : ARRAY[1..GVL_CONSTANTS.C_MAX_BOILERS] OF TON;
  END_VAR

            // Сброс выходов по умолчанию
FOR L_i := 1 TO GVL_CONSTANTS.C_MAX_BOILERS DO
    VO_Boiler_Enable[L_i] := FALSE;
    VO_Boiler_Setpoint[L_i] := 0.0;
END_FOR;

// Инициализация ротации
IF NOT L_Rotation_Initialized THEN
    L_Last_Rotation_MS := VI_System_Time_MS;
    L_Rotation_Initialized := TRUE;
END_IF;

// Принудительная остановка
IF VI_Boiler_Stop THEN
    VO_Lead_Boiler := L_Lead_Boiler;
    RETURN;
END_IF;

// Ротация строго каждые 168 часов
IF (VI_System_Time_MS - L_Last_Rotation_MS) >= L_Rotation_Period_MS THEN
    IF GVL_CONSTANTS.C_MAX_BOILERS > 1 THEN
        L_Lead_Boiler := 3 - L_Lead_Boiler;
    END_IF;
    L_Last_Rotation_MS := VI_System_Time_MS;
END_IF;

L_Reserve_Boiler := SEL(L_Lead_Boiler = 1, 1, 2);

L_Lead_Available :=
    VI_Boiler_OT_Online[L_Lead_Boiler] AND
    NOT VI_Boiler_Error_Status[L_Lead_Boiler];

L_Reserve_Available :=
    (GVL_CONSTANTS.C_MAX_BOILERS > 1) AND
    VI_Boiler_OT_Online[L_Reserve_Boiler] AND
    NOT VI_Boiler_Error_Status[L_Reserve_Boiler];

// Контроль "команда есть, пламени нет" для ведущего котла
L_Flame_Miss_Timer[L_Lead_Boiler](
    IN := VI_Enable AND L_Lead_Available AND NOT VI_DHW_Heating_Demand AND NOT VI_Boiler_Flame_Status[L_Lead_Boiler],
    PT := T#120s
);

IF L_Flame_Miss_Timer[L_Lead_Boiler].Q AND L_Reserve_Available THEN
    L_Lead_Boiler := L_Reserve_Boiler;
    L_Last_Rotation_MS := VI_System_Time_MS;
    L_Lead_Available :=
        VI_Boiler_OT_Online[L_Lead_Boiler] AND
        NOT VI_Boiler_Error_Status[L_Lead_Boiler];
    L_Reserve_Boiler := SEL(L_Lead_Boiler = 1, 1, 2);
    L_Reserve_Available :=
        (GVL_CONSTANTS.C_MAX_BOILERS > 1) AND
        VI_Boiler_OT_Online[L_Reserve_Boiler] AND
        NOT VI_Boiler_Error_Status[L_Reserve_Boiler];
END_IF;

// Нет запроса тепла
IF NOT VI_Enable THEN
    VO_Lead_Boiler := L_Lead_Boiler;
    RETURN;
END_IF;

// Целевая уставка
IF VI_DHW_Heating_Demand THEN
    L_Target_Setpoint := LIMIT(20.0, VI_DHW_Target_Temp + 15.0, 85.0);
ELSE
    L_Target_Setpoint := LIMIT(20.0, VI_Target_Supply_Temp + 5.0, 80.0);
END_IF;

// Выбор ведущего по доступности
IF NOT L_Lead_Available AND L_Reserve_Available THEN
    L_Lead_Boiler := L_Reserve_Boiler;
    L_Lead_Available := TRUE;
    L_Reserve_Boiler := SEL(L_Lead_Boiler = 1, 1, 2);
    L_Reserve_Available :=
        (GVL_CONSTANTS.C_MAX_BOILERS > 1) AND
        VI_Boiler_OT_Online[L_Reserve_Boiler] AND
        NOT VI_Boiler_Error_Status[L_Reserve_Boiler];
END_IF;

// Основной котёл
IF L_Lead_Available THEN
    VO_Boiler_Enable[L_Lead_Boiler] := TRUE;
    VO_Boiler_Setpoint[L_Lead_Boiler] := L_Target_Setpoint;
END_IF;

// Резервный котёл: >80% или отказ основного
L_Start_Reserve :=
    L_Reserve_Available AND
    (
        (VI_Demand_Power > 80.0) OR
        (NOT L_Lead_Available)
    );

IF L_Start_Reserve THEN
    VO_Boiler_Enable[L_Reserve_Boiler] := TRUE;
    VO_Boiler_Setpoint[L_Reserve_Boiler] := L_Target_Setpoint;
END_IF;

VO_Lead_Boiler := L_Lead_Boiler;
          
END_FUNCTION_BLOCK

FUNCTION_BLOCK FB_Trend_Logger
  VAR_INPUT
    VI_System_Time_MS : UDINT;
    VI_Config : ST_Trend_Config;
    VI_Current_Value : REAL;
  END_VAR
  VAR_OUTPUT
    VO_Data : ST_Trend_Data;
  END_VAR
  VAR
    L_Last_Log_Time : UDINT;
    L_Last_Value : REAL;
    L_Deviation : REAL;
    L_Elapsed_Time : UDINT;
    L_Write_Index : UDINT;
  END_VAR

            IF NOT VI_Config.enabled THEN
    RETURN;
END_IF;

L_Deviation := ABS(VI_Current_Value - L_Last_Value);
L_Elapsed_Time := SEL(
    VI_System_Time_MS >= L_Last_Log_Time,
    VI_System_Time_MS - L_Last_Log_Time,
    (4294967295 - L_Last_Log_Time) + VI_System_Time_MS + 1
);

IF (L_Deviation >= (ABS(L_Last_Value) * VI_Config.deviation_threshold_percent / REAL#100.0)) OR
   (L_Elapsed_Time >= GVL_CONSTANTS.C_MS_IN_HOUR) THEN

    L_Write_Index := (VO_Data.record_count MOD 100) + 1;
    VO_Data.write_index := L_Write_Index;
    VO_Data.values[L_Write_Index] := VI_Current_Value;
    VO_Data.timestamps[L_Write_Index] := VI_System_Time_MS;
    VO_Data.record_count := VO_Data.record_count + 1;
    VO_Data.sum_values := VO_Data.sum_values + VI_Current_Value;
    VO_Data.config := VI_Config;

    L_Last_Value := VI_Current_Value;
    L_Last_Log_Time := VI_System_Time_MS;
END_IF;
          
END_FUNCTION_BLOCK

FUNCTION_BLOCK FB_System_Persist_Manager
  VAR_INPUT
    VI_System_Time_MS : UDINT;
    VI_IsActivePLC : BOOL;
  END_VAR
  VAR_IN_OUT
    VIO_Persist_Buffer : ARRAY[0..4] OF BYTE;
    VIO_Last_Written_Persist_Buffer : ARRAY[0..4] OF BYTE;
    VIO_Persist_Buffer_Changed : BOOL;
    VIO_Last_Persist_Write_MS : UDINT;
    VIO_NVRAM_Cmd : BYTE;
    VIO_NVRAM_Offset : UDINT;
    VIO_NVRAM_Done : BOOL;
    VIO_NVRAM_Err : BOOL;
    VIO_NVRAM_ErrID : UDINT;
  END_VAR
  VAR
    fbNVRAMManager : FB_NVRAM_Manager;
  END_VAR

            // ==============================================================================
// System persist manager helper
//
// Internal helper for PRG_System.
// Owns persistent snapshot packing, controlled NVRAM write gating,
// FB_NVRAM_Manager call, and last-written buffer tracking.
// ==============================================================================



// Pack persistent snapshot into compact byte buffer for controlled NVRAM mirroring
VIO_Persist_Buffer[0] := TO_BYTE(TO_INT(GVL_STATE.G_System_Mode));
IF GVL_PERSISTENT.P_Safety_Gas_Latched THEN
    VIO_Persist_Buffer[1] := BYTE#1;
ELSE
    VIO_Persist_Buffer[1] := BYTE#0;
END_IF;
IF GVL_PERSISTENT.P_Safety_Smoke_Latched THEN
    VIO_Persist_Buffer[2] := BYTE#1;
ELSE
    VIO_Persist_Buffer[2] := BYTE#0;
END_IF;
IF GVL_PERSISTENT.P_Safety_Leak_Latched THEN
    VIO_Persist_Buffer[3] := BYTE#1;
ELSE
    VIO_Persist_Buffer[3] := BYTE#0;
END_IF;
IF GVL_PERSISTENT.P_DHW_Heating_Active THEN
    VIO_Persist_Buffer[4] := BYTE#1;
ELSE
    VIO_Persist_Buffer[4] := BYTE#0;
END_IF;

VIO_Persist_Buffer_Changed :=
    (VIO_Persist_Buffer[0] <> VIO_Last_Written_Persist_Buffer[0]) OR
    (VIO_Persist_Buffer[1] <> VIO_Last_Written_Persist_Buffer[1]) OR
    (VIO_Persist_Buffer[2] <> VIO_Last_Written_Persist_Buffer[2]) OR
    (VIO_Persist_Buffer[3] <> VIO_Last_Written_Persist_Buffer[3]) OR
    (VIO_Persist_Buffer[4] <> VIO_Last_Written_Persist_Buffer[4]);

VIO_NVRAM_Cmd := 0;
VIO_NVRAM_Offset := 0;

IF GVL_CONFIG.G_HMI_Apply_Settings THEN
    // explicit config apply may request a controlled write
    VIO_NVRAM_Cmd := 1;
    GVL_CONFIG.G_HMI_Apply_Settings := FALSE;

ELSIF VIO_Persist_Buffer_Changed THEN
    // controlled write: no more often than once per 60 seconds
    IF (VIO_Last_Persist_Write_MS = 0) OR
       ((VI_System_Time_MS - VIO_Last_Persist_Write_MS) >= 60000) THEN
        VIO_NVRAM_Cmd := 1;
    END_IF;
END_IF;

fbNVRAMManager(
    VI_Command := VIO_NVRAM_Cmd,
    VI_Offset := VIO_NVRAM_Offset,
    VI_DataRef := VIO_Persist_Buffer[0],
    VI_DataSize := 5,
    VI_System_Time_MS := VI_System_Time_MS,
    VI_Operator_ID := 'SYSTEM',
    VI_IsActivePLC := VI_IsActivePLC,
    VI_TwoPersonConfirmation := FALSE,
    VO_Done => VIO_NVRAM_Done,
    VO_Error => VIO_NVRAM_Err,
    VO_ErrorID => VIO_NVRAM_ErrID
);

IF (VIO_NVRAM_Cmd = 1) AND VIO_NVRAM_Done AND NOT VIO_NVRAM_Err THEN
    VIO_Last_Written_Persist_Buffer[0] := VIO_Persist_Buffer[0];
    VIO_Last_Written_Persist_Buffer[1] := VIO_Persist_Buffer[1];
    VIO_Last_Written_Persist_Buffer[2] := VIO_Persist_Buffer[2];
    VIO_Last_Written_Persist_Buffer[3] := VIO_Persist_Buffer[3];
    VIO_Last_Written_Persist_Buffer[4] := VIO_Persist_Buffer[4];
    VIO_Last_Persist_Write_MS := VI_System_Time_MS;
END_IF;

// >>> BULK_SYNC_ANCHOR: FB_System_Persist_Manager <<<
          
END_FUNCTION_BLOCK

FUNCTION_BLOCK FB_Runtime_Bus_Replication
  VAR_INPUT
    VI_Enable : BOOL;
    VI_System_Time_MS : UDINT;
  END_VAR
  VAR
    L_Frame : ST_Runtime_Bus_Frame;
    L_TX_Index : UINT;
    L_Finalized_Runtime_Continuity : BOOL;
  END_VAR

            IF NOT VI_Enable THEN
    GVL_Runtime_Bus.G_Runtime_Valid := FALSE;
    RETURN;
END_IF;

L_Finalized_Runtime_Continuity :=
    GVL_SEMANTIC_PROGRESS.Semantic_Forward_Progress_Valid
    AND GVL_SEMANTIC_PROGRESS.Semantic_Execution_Continuity_OK
    AND NOT GVL_SEMANTIC_PROGRESS.Semantic_Progress_Lease_Expired
    AND NOT GVL_SEMANTIC_PROGRESS.Semantic_Progress_Quarantine_Active
    AND GVL_RUNTIME_SNAPSHOT.Snapshot_Frozen
    AND GVL_RUNTIME_SNAPSHOT.Snapshot_Publication_Allowed
    AND GVL_RUNTIME_SNAPSHOT.Snapshot_Copy_Valid
    AND GVL_RUNTIME_SNAPSHOT.Snapshot_Isolation_Valid
    AND NOT GVL_RUNTIME_SNAPSHOT.Snapshot_Mutation_Detected
    AND GVL_DISTRIBUTED_SNAPSHOT.Distributed_Publication_Reconciled
    AND GVL_DISTRIBUTED_SNAPSHOT.Distributed_Publication_Freeze_Valid
    AND GVL_DISTRIBUTED_SNAPSHOT.Distributed_Snapshot_Consistent
    AND GVL_DISTRIBUTED_COMMIT.Distributed_Commit_Valid
    AND GVL_DISTRIBUTED_COMMIT.Publication_Prepare_Valid
    AND GVL_DISTRIBUTED_COMMIT.Publication_Commit_Confirmed
    AND NOT GVL_DISTRIBUTED_COMMIT.Peer_Commit_Mismatch
    AND NOT GVL_DISTRIBUTED_COMMIT.Commit_Lease_Expired
    AND GVL_OUTPUT_EPOCH.Output_Publication_Valid
    AND GVL_OUTPUT_EPOCH.Output_Runtime_Epoch_Valid
    AND NOT GVL_OUTPUT_EPOCH.Output_Lease_Expired
    AND NOT GVL_OUTPUT_EPOCH.Output_Forced_Safe_Decay
    AND GVL_COMMAND_VERIFY.PreOutput_Barrier_OK
    AND NOT GVL_COMMAND_VERIFY.PreOutput_Block_IO;

L_TX_Index := UDINT_TO_UINT(GVL_Runtime_Bus.G_Last_Sequence_Id + 1);

IF L_TX_Index > 128 THEN
    L_TX_Index := 1;
END_IF;

L_Frame.Frame_Valid := TRUE;

L_Frame.Frame_Time_MS := VI_System_Time_MS;
L_Frame.Frame_Id := GVL_Runtime_Bus.G_Last_Frame_Id + 1;

L_Frame.Source_Controller_Id :=
    GVL_Distributed_Runtime.G_Local_Node_State.Controller_Id;

L_Frame.Source_Runtime_Node_Id :=
    GVL_Distributed_Runtime.G_Local_Node_State.Runtime_Node_Id;

L_Frame.Frame_Sequence_Id :=
    GVL_Runtime_Bus.G_Last_Sequence_Id + 1;

L_Frame.Frame_Ack_Required := TRUE;

L_Frame.Authority_State_Frame := TRUE;
L_Frame.Recovery_State_Frame := TRUE;
L_Frame.Quarantine_State_Frame := TRUE;
L_Frame.Topology_State_Frame := TRUE;
L_Frame.Binding_State_Frame := TRUE;
L_Frame.Predictive_State_Frame := TRUE;

IF GVL_Distributed_Authority.G_Distributed_Safety_Barrier_OK
   AND NOT GVL_Distributed_Runtime.G_Split_Brain_Suspected
   AND L_Finalized_Runtime_Continuity THEN

    L_Frame.Replication_Consistent := TRUE;

    L_Frame.Status_Code := 0;
    L_Frame.Status_Text :=
        'Deterministic replication frame accepted';

ELSE

    L_Frame.Replication_Rejected := TRUE;

    L_Frame.Status_Code := 2;
    L_Frame.Status_Text :=
        'Deterministic replication frame rejected';

END_IF;

GVL_Runtime_Bus.G_TX_Frames[L_TX_Index] := L_Frame;

GVL_Runtime_Bus.G_Last_Frame_Id :=
    L_Frame.Frame_Id;

GVL_Runtime_Bus.G_Last_Sequence_Id :=
    L_Frame.Frame_Sequence_Id;

GVL_Runtime_Bus.G_TX_Healthy :=
    L_Frame.Replication_Consistent;

GVL_Runtime_Bus.G_RX_Healthy := TRUE;

GVL_Runtime_Bus.G_Any_Replication_Rejected :=
    L_Frame.Replication_Rejected;

GVL_Runtime_Bus.G_Runtime_Valid := TRUE;
GVL_Runtime_Bus.G_Last_Update_MS := VI_System_Time_MS;

IF L_Frame.Replication_Rejected THEN
    GVL_Runtime_Bus.G_Status_Code := 2;
    GVL_Runtime_Bus.G_Status_Text :=
        'Runtime bus replication rejected';
ELSE
    GVL_Runtime_Bus.G_Status_Code := 0;
    GVL_Runtime_Bus.G_Status_Text :=
        'Runtime bus replication healthy';
END_IF;
          
END_FUNCTION_BLOCK

FUNCTION_BLOCK FB_State_Manager
  VAR_INPUT
    VI_System_Severity : E_System_Severity;
    VI_Root_Cause : E_System_Root_Cause;
    VI_Freeze_Risk : BOOL := FALSE;
  END_VAR
  VAR_OUTPUT
    VO_System_OK : BOOL;
    VO_System_Warning : BOOL;
    VO_System_Critical : BOOL;
    VO_Status_Msg : STRING(200);
    VO_System_Mode : E_System_Operating_Mode;
  END_VAR
  VAR
    L_Requested_Mode : E_System_Operating_Mode;
  END_VAR

            VO_System_OK := FALSE;
VO_System_Warning := FALSE;
VO_System_Critical := FALSE;
VO_Status_Msg := '';

// ------------------------------------------------------
// Stateful deterministic mode governance.
// ------------------------------------------------------
// SAFE_STOP entry is immediate.
// SAFE_STOP exit is convergence-lease gated.
//
// Prevents one-cycle false recovery and transient
// healthy visibility from restoring system operation.
// ------------------------------------------------------

L_Requested_Mode := E_System_Operating_Mode.MODE_NORMAL;

CASE VI_System_Severity OF
    E_System_Severity.SEV_NORMAL:
        VO_System_OK := TRUE;
        VO_Status_Msg := 'Система в норме';
        L_Requested_Mode := E_System_Operating_Mode.MODE_NORMAL;

    E_System_Severity.SEV_WARNING:
        VO_System_Warning := TRUE;
        L_Requested_Mode := E_System_Operating_Mode.MODE_DEGRADED;

        CASE VI_Root_Cause OF
            E_System_Root_Cause.ROOT_WATER_LEAK:
                VO_Status_Msg := 'Предупреждение: протечка воды';

            E_System_Root_Cause.ROOT_CO_WARNING:
                VO_Status_Msg := 'Предупреждение: повышенный CO';

            ELSE
                VO_Status_Msg := 'Предупреждение системы';
        END_CASE;

    E_System_Severity.SEV_DEGRADED:
        VO_System_Warning := TRUE;
        L_Requested_Mode := E_System_Operating_Mode.MODE_DEGRADED;

        CASE VI_Root_Cause OF
            E_System_Root_Cause.ROOT_SENSOR_FAULT:
                VO_Status_Msg := 'Деградация: ошибка датчика';

            E_System_Root_Cause.ROOT_IO_OFFLINE:
                VO_Status_Msg := 'Деградация: модуль IO недоступен';

            E_System_Root_Cause.ROOT_COMM_FAULT:
                VO_Status_Msg := 'Деградация: ошибка связи';

            E_System_Root_Cause.ROOT_WATCHDOG_FAULT:
                VO_Status_Msg := 'Деградация: watchdog fault';

            E_System_Root_Cause.ROOT_SUBSYSTEM_FAULT:
                VO_Status_Msg := 'Деградация: ошибка подсистемы';

            ELSE
                VO_Status_Msg := 'Деградация системы';
        END_CASE;

    E_System_Severity.SEV_CRITICAL:
        VO_System_Critical := TRUE;

        IF (VI_Root_Cause = E_System_Root_Cause.ROOT_GAS_LEAK OR
            VI_Root_Cause = E_System_Root_Cause.ROOT_CO_CRITICAL) AND
            VI_Freeze_Risk THEN
            L_Requested_Mode := E_System_Operating_Mode.MODE_FREEZE_PROTECTION;
        ELSE
            L_Requested_Mode := E_System_Operating_Mode.MODE_SAFE_STOP;
        END_IF;

        CASE VI_Root_Cause OF
            E_System_Root_Cause.ROOT_FIRE:
                VO_Status_Msg := 'АВАРИЯ: ПОЖАР';

            E_System_Root_Cause.ROOT_GAS_LEAK:
                VO_Status_Msg := 'АВАРИЯ: УТЕЧКА ГАЗА';

            E_System_Root_Cause.ROOT_CO_CRITICAL:
                VO_Status_Msg := 'АВАРИЯ: КРИТИЧЕСКИЙ CO';

            E_System_Root_Cause.ROOT_WATCHDOG_FAULT:
                VO_Status_Msg := 'АВАРИЯ: WATCHDOG';

            ELSE
                VO_Status_Msg := 'АВАРИЯ СИСТЕМЫ';
        END_CASE;
END_CASE;

// ------------------------------------------------------
// Deterministic SAFE_STOP exit hardening.
// ------------------------------------------------------
// SAFE_STOP/FREEZE_PROTECTION exit requires sustained
// convergence evidence and convergence lease acquisition.
// ------------------------------------------------------

IF (VO_System_Mode = E_System_Operating_Mode.MODE_SAFE_STOP)
OR (VO_System_Mode = E_System_Operating_Mode.MODE_FREEZE_PROTECTION)
THEN
    IF (L_Requested_Mode <> E_System_Operating_Mode.MODE_SAFE_STOP)
    AND (L_Requested_Mode <> E_System_Operating_Mode.MODE_FREEZE_PROTECTION)
    THEN
        IF NOT GVL_CONVERGENCE.Convergence_Lease_OK THEN
            // Hold previous safe mode until deterministic
            // convergence/recovery proof exists.
            L_Requested_Mode := VO_System_Mode;

            IF VO_Status_Msg = '' THEN
                VO_Status_Msg := 'Ожидание подтверждения восстановления';
            ELSE
                VO_Status_Msg := CONCAT(VO_Status_Msg, ' | convergence pending');
            END_IF;
        END_IF;
    END_IF;
END_IF;

VO_System_Mode := L_Requested_Mode;

// >>> BULK_SYNC_ANCHOR: FB_State_Manager <<<
          
END_FUNCTION_BLOCK

FUNCTION_BLOCK FB_Water_Leak_Runtime_Projection
  VAR_INPUT
    VI_Enable : BOOL;
    VI_System_Time_MS : UDINT;
  END_VAR
  VAR
    L_i : INT;
    L_Runtime_State : ST_Water_Leak_Runtime_State;
    L_Global_Leak : BOOL;
    L_Global_Warning : BOOL;
  END_VAR

            IF NOT VI_Enable THEN
    GVL_Water_Runtime_Projection.G_Projection_Valid := FALSE;
    RETURN;
END_IF;

L_Global_Leak := FALSE;
L_Global_Warning := FALSE;

FOR L_i := 1 TO GVL_CONSTANTS.C_MAX_FLOOD_SENSORS DO

    L_Runtime_State.Projection_Valid := FALSE;
    L_Runtime_State.Projection_Valid := TRUE;
    L_Runtime_State.Projection_System_Time_MS := VI_System_Time_MS;
    L_Runtime_State.Physical_Sensor_Index := TO_UINT(L_i);
    L_Runtime_State.Physical_Input_Valid := TRUE;
    L_Runtime_State.Leak_Warning_Active := GVL_STATE.G_Flood_Warning[L_i];
    L_Runtime_State.Leak_Confirmed := GVL_STATE.G_Flood_Alarm[L_i];
    L_Runtime_State.Active_Safety_Leak_Latched := GVL_INTENT_SAFETY.I_Water_Main_Close_Required;
    L_Runtime_State.Active_Global_Close_Path := GVL_COMMAND_SHADOW.G_Close_Valve_35 OR GVL_COMMAND_SHADOW.G_Close_Valve_36;

    L_Runtime_State.Mapping_Valid := (GVL_CONFIG.G_Flood_Global_Config.sensor_to_valve_map[L_i] <> 0);
    L_Runtime_State.Mapping_Missing := NOT L_Runtime_State.Mapping_Valid;

    IF L_Runtime_State.Mapping_Valid THEN
        L_Runtime_State.Valve_Group_Id := TO_UINT(GVL_CONFIG.G_Flood_Global_Config.sensor_to_valve_map[L_i]);
        L_Runtime_State.Selective_Isolation_Possible := TRUE;
        L_Runtime_State.Fallback_Global_Isolation_Required := FALSE;
    ELSE
        L_Runtime_State.Selective_Isolation_Possible := FALSE;
        L_Runtime_State.Fallback_Global_Isolation_Required := TRUE;
    END_IF;

    L_Runtime_State.Logical_Sensor_Valid := TRUE;
    L_Runtime_State.Hydraulic_Zone_Id := TO_UINT(L_i);
    L_Runtime_State.Hydraulic_Segment_Id := TO_UINT(L_i);
    L_Runtime_State.Isolation_Group_Id := L_Runtime_State.Valve_Group_Id;

    IF L_Runtime_State.Leak_Confirmed THEN
        L_Runtime_State.Leak_Confidence := 1.0;
    ELSIF L_Runtime_State.Leak_Warning_Active THEN
        L_Runtime_State.Leak_Confidence := 0.5;
    ELSE
        L_Runtime_State.Leak_Confidence := 0.0;
    END_IF;

    L_Runtime_State.Sensor_Quality_Valid := TRUE;

    IF L_Runtime_State.Leak_Confirmed THEN
        IF L_Runtime_State.Mapping_Valid THEN
            L_Runtime_State.Reason_Code := 1;
            L_Runtime_State.Reason_Text := 'Leak confirmed';
        ELSE
            L_Runtime_State.Reason_Code := 2;
            L_Runtime_State.Reason_Text := 'Leak confirmed fallback';
        END_IF;
    ELSIF L_Runtime_State.Leak_Warning_Active THEN
        L_Runtime_State.Reason_Code := 3;
        L_Runtime_State.Reason_Text := 'Leak warning active';
    ELSE
        L_Runtime_State.Reason_Code := 0;
        L_Runtime_State.Reason_Text := 'No leak activity';
    END_IF;

    L_Runtime_State.Warning_Started_Event := GVL_STATE.G_Flood_Warning_Rise[L_i];
    L_Runtime_State.Leak_Confirmed_Event := GVL_STATE.G_Flood_Alarm_Rise[L_i];
    L_Runtime_State.Leak_Cleared_Event := GVL_STATE.G_Flood_Alarm_Fall[L_i];
    L_Runtime_State.Isolation_Requested_Event := L_Runtime_State.Leak_Confirmed;
    L_Runtime_State.Mapping_Invalid_Event := L_Runtime_State.Mapping_Missing;
    L_Runtime_State.Supervisory_Observation_Only := TRUE;

    GVL_Water_Runtime_Projection.G_Leak_Runtime_State[L_i] := L_Runtime_State;

    L_Global_Leak := L_Global_Leak OR L_Runtime_State.Leak_Confirmed;
    L_Global_Warning := L_Global_Warning OR L_Runtime_State.Leak_Warning_Active;
END_FOR;

GVL_Water_Runtime_Projection.G_Global_Leak_Active := L_Global_Leak;
GVL_Water_Runtime_Projection.G_Global_Warning_Active := L_Global_Warning;
GVL_Water_Runtime_Projection.G_Projection_Valid := TRUE;
GVL_Water_Runtime_Projection.G_Last_Projection_MS := VI_System_Time_MS;
GVL_Water_Runtime_Projection.G_Runtime_Projection_Status_Code := 0;
GVL_Water_Runtime_Projection.G_Runtime_Projection_Status_Text := 'Water runtime semantic projection active';
          
END_FUNCTION_BLOCK

FUNCTION_BLOCK FB_Heating_System_Manager
  VAR_INPUT
    VI_System_Mode : E_System_Operating_Mode;
    VI_System_Time_MS : UDINT;
    VI_IsActivePLC : BOOL;
    VI_Outdoor_Temp : REAL;
    VI_Config : ST_Heating_Config;
    VI_Tariff : ST_Tariff_Config;
    VI_Current_Hour : UINT;
    VI_DHW_Heating_Demand : BOOL;
    VI_DHW_Target_Temp : REAL;
    VI_Emergency_Stop : BOOL;
    VI_Gas_Safety_Stop : BOOL;
    VI_Boiler_Error_Status : ARRAY[1..GVL_CONSTANTS.C_MAX_BOILERS] OF BOOL;
    VI_Boiler_OT_Online : ARRAY[1..GVL_CONSTANTS.C_MAX_BOILERS] OF BOOL;
    VI_Boiler_Modulation : ARRAY[1..GVL_CONSTANTS.C_MAX_BOILERS] OF REAL;
  END_VAR
  VAR_OUTPUT
    VO_Manifold_Valves : ARRAY[1..GVL_CONSTANTS.C_MAX_MANIFOLDS] OF REAL;
    VO_Manifold_Pumps : ARRAY[1..GVL_CONSTANTS.C_MAX_MANIFOLDS] OF BOOL;
    VO_Zone_Valves : ARRAY[1..GVL_CONSTANTS.C_MAX_HEATING_CIRCUITS] OF BOOL;
    VO_Boiler_OT_Enable : ARRAY[1..GVL_CONSTANTS.C_MAX_BOILERS] OF BOOL;
    VO_Boiler_OT_Setpoint : ARRAY[1..GVL_CONSTANTS.C_MAX_BOILERS] OF REAL;
    VO_Backup_Circulation_Pump : BOOL;
    VO_Electric_Heater_Enable : BOOL;
    VO_Freeze_Risk_Status : BOOL;
    VO_Status : ARRAY[1..GVL_CONSTANTS.C_MAX_MANIFOLDS] OF ST_Manifold_Status;
    VO_Boiler_Status : ARRAY[1..GVL_CONSTANTS.C_MAX_BOILERS] OF ST_Boiler_Status;
  END_VAR
  VAR_IN_OUT
    VI_Floor_Temps : ARRAY[1..GVL_CONSTANTS.C_MAX_HEATING_CIRCUITS] OF REAL;
    VI_Room_Temps : ARRAY[1..GVL_CONSTANTS.C_MAX_ZONES] OF REAL;
    VI_Manifold_Pressures : ARRAY[1..GVL_CONSTANTS.C_MAX_MANIFOLDS] OF REAL;
    VI_Manifold_Currents : ARRAY[1..GVL_CONSTANTS.C_MAX_MANIFOLDS] OF REAL;
    VI_Manifold_Temps_Supply : ARRAY[1..GVL_CONSTANTS.C_MAX_MANIFOLDS] OF REAL;
    VI_Manifold_Temps_Return : ARRAY[1..GVL_CONSTANTS.C_MAX_MANIFOLDS] OF REAL;
    VI_Boiler_Flame_Status : ARRAY[1..GVL_CONSTANTS.C_MAX_BOILERS] OF BOOL;
    VI_Zone_Configs : ARRAY[1..GVL_CONSTANTS.C_MAX_HEATING_CIRCUITS] OF ST_FloorHeating_Circuit_Config;
    VI_Rule_Actions : ARRAY[1..GVL_CONSTANTS.C_MAX_RULES] OF ST_Rule_Action;
    VI_IO_Modules_Online : ARRAY[1..GVL_CONSTANTS.C_MAX_MODULES] OF BOOL;
    VI_Manifold_End_Switches : ARRAY[1..GVL_CONSTANTS.C_MAX_MANIFOLDS] OF BOOL;
    VI_Valve_Test_Config : ARRAY[1..GVL_CONSTANTS.C_MAX_MANIFOLDS] OF ST_Valve_Test_Config;
  END_VAR
  VAR
    L_i : INT;
    L_Target_Supply_Temp : REAL;
    L_Manifold_Demand_Map : ARRAY[1..GVL_CONSTANTS.C_MAX_MANIFOLDS] OF BOOL;
    L_Manifold_Demand_Filtered : ARRAY[1..GVL_CONSTANTS.C_MAX_MANIFOLDS] OF BOOL;
    L_Manifold_Available : ARRAY[1..GVL_CONSTANTS.C_MAX_MANIFOLDS] OF BOOL;
    L_Manifold_In_Service : ARRAY[1..GVL_CONSTANTS.C_MAX_MANIFOLDS] OF BOOL;
    L_Manifold_Subsystem_Degraded : ARRAY[1..GVL_CONSTANTS.C_MAX_MANIFOLDS] OF BOOL;
    L_Manifold_Base_Priority : ARRAY[1..GVL_CONSTANTS.C_MAX_MANIFOLDS] OF INT;
    L_Manifold_Effective_Priority : ARRAY[1..GVL_CONSTANTS.C_MAX_MANIFOLDS] OF INT;
    L_Manifold_Thermal_Weight : ARRAY[1..GVL_CONSTANTS.C_MAX_MANIFOLDS] OF REAL;
    L_Allocation_Degraded : BOOL;
    fbValveTestManager : FB_Valve_Test_Manager;
    L_IO_Failsafe_Active : BOOL;
    L_Freeze_Active : BOOL;
    L_Freeze_Target_Supply : REAL;
    L_Policy_Degraded : BOOL;
    L_Sensor_Error : BOOL;
    L_Subsys_Degraded : BOOL;
    L_Pressure_OK : BOOL;
    L_Prev_Pressure : ARRAY[1..GVL_CONSTANTS.C_MAX_MANIFOLDS] OF REAL;
    L_Prev_Current : ARRAY[1..GVL_CONSTANTS.C_MAX_MANIFOLDS] OF REAL;
    L_Confidence : REAL;
    L_Policy_Target_Adjustment : REAL;
    fbAdaptiveTarget : FB_Heating_Adaptive_Target;
    fbSafetyGate : FB_Heating_Safety_Gate;
    fbSafeState : FB_Heating_Safe_State;
    fbDemandMap : FB_Heating_Demand_Map;
    fbPolicyPriorityBridge : FB_Heating_Policy_Priority_Bridge;
    fbAllocationFilter : FB_Heating_Allocation_Filter;
    fbRuntimeObservability : FB_Heating_Runtime_Observability;
    fbCircuitControl : FB_Heating_Circuit_Control;
    fbManifoldControl : FB_Heating_Manifold_Control;
    fbBoilerControl : FB_Heating_Boiler_Control;
  END_VAR

            L_Policy_Degraded := (VI_System_Mode = E_System_Operating_Mode.MODE_DEGRADED);

GVL_STATE.G_Heating_IO_Fault := FALSE;
GVL_STATE.G_Heating_Sensor_Fault := FALSE;
GVL_STATE.G_Heating_Subsystem_Degraded := FALSE;
L_Sensor_Error := FALSE;
L_Subsys_Degraded := FALSE;
L_Allocation_Degraded := FALSE;

L_IO_Failsafe_Active := FALSE;
FOR L_i := 1 TO GVL_CONSTANTS.C_MAX_MODULES DO
    IF NOT VI_IO_Modules_Online[L_i] THEN
        L_IO_Failsafe_Active := TRUE;
        GVL_STATE.G_Heating_IO_Fault := TRUE;
        GVL_STATE.G_Heating_Subsystem_Degraded := TRUE;
        EXIT;
    END_IF;
END_FOR;

fbSafetyGate(
    VI_System_Mode := VI_System_Mode,
    VI_Emergency_Stop := VI_Emergency_Stop,
    VI_Gas_Safety_Stop := VI_Gas_Safety_Stop,
    VI_IO_Failsafe_Active := L_IO_Failsafe_Active,
    VI_Outdoor_Temp := VI_Outdoor_Temp,
    VI_Freeze_Threshold := VI_Config.Freeze_Threshold,
    VI_Floor_Temps := VI_Floor_Temps,
    VO_Freeze_Mode_Active => L_Freeze_Active,
    VO_Freeze_Target_Supply => L_Freeze_Target_Supply
);

fbSafeState(
    VI_Block_Normal_Heating := fbSafetyGate.VO_Block_Normal_Heating,
    VI_IO_Failsafe_Active := fbSafetyGate.VO_IO_Failsafe_Active,
    VI_Gas_Safety_Active := fbSafetyGate.VO_Gas_Safety_Active,
    VI_Freeze_Active := L_Freeze_Active,
    VI_Freeze_Target_Supply := L_Freeze_Target_Supply,
    VI_Manifold_Temps_Supply := VI_Manifold_Temps_Supply,
    VI_Boiler_Error_Status := VI_Boiler_Error_Status,
    VI_Boiler_OT_Online := VI_Boiler_OT_Online
);

IF fbSafeState.VO_Applied THEN
    FOR L_i := 1 TO GVL_CONSTANTS.C_MAX_HEATING_CIRCUITS DO
        VO_Zone_Valves[L_i] := fbSafeState.VO_Zone_Valves[L_i];
    END_FOR;

    FOR L_i := 1 TO GVL_CONSTANTS.C_MAX_MANIFOLDS DO
        VO_Manifold_Pumps[L_i] := fbSafeState.VO_Manifold_Pumps[L_i];
        VO_Manifold_Valves[L_i] := fbSafeState.VO_Manifold_Valves[L_i];
    END_FOR;

    FOR L_i := 1 TO GVL_CONSTANTS.C_MAX_BOILERS DO
        VO_Boiler_OT_Enable[L_i] := fbSafeState.VO_Boiler_OT_Enable[L_i];
        VO_Boiler_OT_Setpoint[L_i] := fbSafeState.VO_Boiler_OT_Setpoint[L_i];
        VO_Boiler_Status[L_i] := fbSafeState.VO_Boiler_Status[L_i];
    END_FOR;

    VO_Backup_Circulation_Pump := fbSafeState.VO_Backup_Circulation_Pump;
    VO_Electric_Heater_Enable := fbSafeState.VO_Electric_Heater_Enable;
    VO_Freeze_Risk_Status := fbSafeState.VO_Freeze_Risk_Status;
    RETURN;
END_IF;

VO_Backup_Circulation_Pump := FALSE;
VO_Electric_Heater_Enable := FALSE;
VO_Freeze_Risk_Status := FALSE;

IF L_Freeze_Active THEN
    L_Target_Supply_Temp := L_Freeze_Target_Supply;
ELSE
    L_Target_Supply_Temp := VI_Config.Target_Floor_Temp;
END_IF;

fbAdaptiveTarget(
    VI_Base_Target_Supply_Temp := L_Target_Supply_Temp,
    VI_Global_Target_Temperature := GVL_STATE.G_Target_Temperature,
    VI_Zone_Configs := VI_Zone_Configs,
    VI_Floor_Temps := VI_Floor_Temps,
    VI_Room_Temps := VI_Room_Temps,
    VO_Target_Supply_Temp => L_Target_Supply_Temp
);

L_Policy_Target_Adjustment := GVL_HEATING_POLICY.G_Policy_Target_Adjustment;

IF L_Policy_Target_Adjustment > REAL#5.0 THEN
    L_Policy_Target_Adjustment := REAL#5.0;
ELSIF L_Policy_Target_Adjustment < REAL#-3.0 THEN
    L_Policy_Target_Adjustment := REAL#-3.0;
END_IF;

L_Target_Supply_Temp :=
    LIMIT(
        GVL_CONSTANTS.C_BOILER_SETPOINT_MIN,
        L_Target_Supply_Temp + L_Policy_Target_Adjustment,
        GVL_CONSTANTS.C_BOILER_SETPOINT_MAX
    );

fbCircuitControl(
    VI_System_Time_MS := VI_System_Time_MS,
    VI_Current_Hour := VI_Current_Hour,
    VI_IsActivePLC := VI_IsActivePLC,
    VI_Config := VI_Config,
    VI_Tariff := VI_Tariff,
    VI_Scenario_Adjust := REAL#0.0,
    VI_Zone_Configs := VI_Zone_Configs,
    VI_Floor_Temps := VI_Floor_Temps,
    VI_Room_Temps := VI_Room_Temps,
    VI_Rule_Actions := VI_Rule_Actions,
    VO_Zone_Valves => VO_Zone_Valves,
    VO_Heating_Sensor_Fault => L_Sensor_Error
);

GVL_STATE.G_Heating_Sensor_Fault := L_Sensor_Error;

fbDemandMap(
    VI_Zone_Valves := VO_Zone_Valves,
    VI_Zone_Configs := VI_Zone_Configs,
    VO_Manifold_Demand_Map => L_Manifold_Demand_Map
);

FOR L_i := 1 TO GVL_CONSTANTS.C_MAX_MANIFOLDS DO
    L_Manifold_Available[L_i] := VI_Manifold_Pressures[L_i] >= GVL_CONSTANTS.C_MIN_HEATING_MANIFOLD_PRESSURE;
    L_Manifold_In_Service[L_i] := GVL_CONFIG.G_Manifold_Pump_In_Service[L_i];
    L_Manifold_Subsystem_Degraded[L_i] :=
        GVL_STATE.G_Predictive_Pump_Pressure_Drop[L_i]
        OR GVL_STATE.G_Predictive_Pump_Current_Rise[L_i];

    L_Manifold_Base_Priority[L_i] := GVL_CONFIG.G_Manifold_Priority[L_i];
    L_Manifold_Thermal_Weight[L_i] := GVL_CONFIG.G_Manifold_Thermal_Weight[L_i];
END_FOR;

fbPolicyPriorityBridge(
    VI_Enable := (GVL_CONFIG.G_Max_Thermal_Budget > REAL#0.0),
    VI_Zone_Valves := VO_Zone_Valves,
    VI_Zone_Configs := VI_Zone_Configs,
    VI_Manifold_Base_Priority := L_Manifold_Base_Priority,
    VI_Zone_Priority_Bias := GVL_HEATING_POLICY.G_Zone_Priority_Bias,
    VI_Policy_Priority_Multiplier := GVL_HEATING_POLICY.G_Policy_Priority_Multiplier,
    VO_Manifold_Effective_Priority => L_Manifold_Effective_Priority
);

fbAllocationFilter(
    VI_Enable := TRUE,
    VI_Enable_Policy_Allocation := (GVL_CONFIG.G_Max_Thermal_Budget > REAL#0.0),
    VI_Freeze_Mode_Active := L_Freeze_Active,
    VI_DHW_Heating_Demand := VI_DHW_Heating_Demand,
    VI_Manifold_Demand_Map := L_Manifold_Demand_Map,
    VI_Manifold_Available := L_Manifold_Available,
    VI_Manifold_In_Service := L_Manifold_In_Service,
    VI_Manifold_Subsystem_Degraded := L_Manifold_Subsystem_Degraded,
    VI_Manifold_Base_Priority := L_Manifold_Effective_Priority,
    VI_Manifold_Thermal_Weight := L_Manifold_Thermal_Weight,
    VI_Max_Thermal_Budget := GVL_CONFIG.G_Max_Thermal_Budget,
    VO_Manifold_Demand_Filtered => L_Manifold_Demand_Filtered,
    VO_Allocation_Degraded => L_Allocation_Degraded
);

fbRuntimeObservability(
    VI_Policy_Active := (GVL_CONFIG.G_Max_Thermal_Budget > REAL#0.0),
    VI_Freeze_Bypass_Active := L_Freeze_Active,
    VI_DHW_Bypass_Active := VI_DHW_Heating_Demand,
    VI_Budget_Max := GVL_CONFIG.G_Max_Thermal_Budget,
    VI_Budget_Used := fbAllocationFilter.VO_Thermal_Budget_Used,
    VI_Requested := L_Manifold_Demand_Map,
    VI_Allowed := fbAllocationFilter.VO_Manifold_Allowed,
    VI_Filtered := L_Manifold_Demand_Filtered,
    VI_Block_Reason := fbAllocationFilter.VO_Manifold_Block_Reason,
    VI_Effective_Priority := fbAllocationFilter.VO_Manifold_Priority_Effective,
    VI_Priority_Bridge_Active := fbPolicyPriorityBridge.VO_Bridge_Active,
    VI_Priority_Bias_Applied := fbPolicyPriorityBridge.VO_Manifold_Priority_Bias_Applied,
    VI_Priority_Effective := L_Manifold_Effective_Priority
);

IF L_Allocation_Degraded THEN
    GVL_STATE.G_Heating_Subsystem_Degraded := TRUE;
END_IF;

fbManifoldControl(
    VI_System_Time_MS := VI_System_Time_MS,
    VI_IsActivePLC := VI_IsActivePLC,
    VI_DHW_Heating_Demand := VI_DHW_Heating_Demand,
    VI_Freeze_Mode_Active := L_Freeze_Active,
    VI_Target_Supply_Temp := L_Target_Supply_Temp,
    VI_Any_Zone_Active := L_Manifold_Demand_Filtered,
    VI_Manifold_Pressures := VI_Manifold_Pressures,
    VI_Manifold_Currents := VI_Manifold_Currents,
    VI_Manifold_Temps_Supply := VI_Manifold_Temps_Supply,
    VI_Manifold_Temps_Return := VI_Manifold_Temps_Return,
    VO_Manifold_Pumps => VO_Manifold_Pumps,
    VO_Manifold_Valves => VO_Manifold_Valves,
    VO_Status => VO_Status
);

FOR L_i := 1 TO GVL_CONSTANTS.C_MAX_MANIFOLDS DO
    L_Pressure_OK := VI_Manifold_Pressures[L_i] >= GVL_CONSTANTS.C_MIN_HEATING_MANIFOLD_PRESSURE;

    IF VO_Manifold_Pumps[L_i] AND NOT L_Pressure_OK THEN
        VO_Manifold_Pumps[L_i] := FALSE;
        GVL_STATE.G_Heating_Subsystem_Degraded := TRUE;
    END_IF;

    IF (L_Prev_Pressure[L_i] > REAL#0.0) AND ((L_Prev_Pressure[L_i] - VI_Manifold_Pressures[L_i]) > REAL#0.2) THEN
        GVL_STATE.G_Predictive_Pump_Pressure_Drop[L_i] := TRUE;
    ELSE
        GVL_STATE.G_Predictive_Pump_Pressure_Drop[L_i] := FALSE;
    END_IF;

    IF (L_Prev_Current[L_i] > REAL#0.0) AND (VI_Manifold_Currents[L_i] > (L_Prev_Current[L_i] * REAL#1.2)) THEN
        GVL_STATE.G_Predictive_Pump_Current_Rise[L_i] := TRUE;
    ELSE
        GVL_STATE.G_Predictive_Pump_Current_Rise[L_i] := FALSE;
    END_IF;

    IF GVL_STATE.G_Predictive_Pump_Pressure_Drop[L_i] OR GVL_STATE.G_Predictive_Pump_Current_Rise[L_i] THEN
        GVL_STATE.G_Heating_Subsystem_Degraded := TRUE;
    END_IF;

    L_Prev_Pressure[L_i] := VI_Manifold_Pressures[L_i];
    L_Prev_Current[L_i] := VI_Manifold_Currents[L_i];
END_FOR;

// ======================================================
// HEATING CONFIDENCE PUBLICATION
// ======================================================
// The former local error-score decay path has been replaced by the
// normalized input confidence surface. Runtime faults may still reduce
// confidence and reason publication, but the base confidence now comes
// from canonical input semantics.
L_Confidence := GVL_INPUT.IN_Min_Zone_Confidence;

IF L_Confidence < REAL#0.0 THEN
    L_Confidence := REAL#0.0;
ELSIF L_Confidence > REAL#1.0 THEN
    L_Confidence := REAL#1.0;
END_IF;

GVL_STATE.G_Heating_Confidence_Reason_Code := 0;
GVL_STATE.G_Heating_Confidence_Reason_Text := 'OK';

IF GVL_INPUT.IN_Input_Degraded OR GVL_INPUT.IN_Anomaly_Detected THEN
    GVL_STATE.G_Heating_Subsystem_Degraded := TRUE;
    GVL_STATE.G_Heating_Confidence_Reason_Code := 5;

    IF GVL_INPUT.IN_Anomaly_Reason <> '' THEN
        GVL_STATE.G_Heating_Confidence_Reason_Text := GVL_INPUT.IN_Anomaly_Reason;
    ELSE
        GVL_STATE.G_Heating_Confidence_Reason_Text := 'Input quality degraded';
    END_IF;
END_IF;

IF GVL_STATE.G_Heating_IO_Fault THEN
    IF L_Confidence > REAL#0.8 THEN
        L_Confidence := REAL#0.8;
    END_IF;
    GVL_STATE.G_Heating_Confidence_Reason_Code := 2;
    GVL_STATE.G_Heating_Confidence_Reason_Text := 'IO fault detected';
ELSIF GVL_STATE.G_Heating_Sensor_Fault THEN
    IF L_Confidence > REAL#0.6 THEN
        L_Confidence := REAL#0.6;
    END_IF;
    GVL_STATE.G_Heating_Confidence_Reason_Code := 1;
    GVL_STATE.G_Heating_Confidence_Reason_Text := 'Sensor fault detected';
ELSE
    FOR L_i := 1 TO GVL_CONSTANTS.C_MAX_MANIFOLDS DO
        IF VI_Manifold_Pressures[L_i] < GVL_CONSTANTS.C_MIN_HEATING_MANIFOLD_PRESSURE THEN
            IF L_Confidence > REAL#0.7 THEN
                L_Confidence := REAL#0.7;
            END_IF;
            GVL_STATE.G_Heating_Confidence_Reason_Code := 3;
            GVL_STATE.G_Heating_Confidence_Reason_Text := 'Low manifold pressure';
            EXIT;
        END_IF;
    END_FOR;

    FOR L_i := 1 TO GVL_CONSTANTS.C_MAX_MANIFOLDS DO
        IF GVL_STATE.G_Predictive_Pump_Pressure_Drop[L_i] OR GVL_STATE.G_Predictive_Pump_Current_Rise[L_i] THEN
            IF L_Confidence > REAL#0.75 THEN
                L_Confidence := REAL#0.75;
            END_IF;
            GVL_STATE.G_Heating_Confidence_Reason_Code := 4;
            GVL_STATE.G_Heating_Confidence_Reason_Text := 'Predictive pump degradation';
            EXIT;
        END_IF;
    END_FOR;
END_IF;

GVL_STATE.G_Heating_Confidence := L_Confidence;
GVL_STATE.G_Heating_Error_Score := REAL#1.0 - L_Confidence;

IF GVL_STATE.G_Heating_Confidence < REAL#0.5 THEN
    L_Target_Supply_Temp := L_Target_Supply_Temp - REAL#3.0;
END_IF;

CASE GVL_STATE.G_Heating_Confidence_Reason_Code OF
    1:
        L_Target_Supply_Temp := LIMIT(GVL_CONSTANTS.C_BOILER_SETPOINT_MIN, REAL#40.0, GVL_CONSTANTS.C_BOILER_SETPOINT_MAX);
    2:
        VO_Backup_Circulation_Pump := TRUE;
    3:
        FOR L_i := 1 TO GVL_CONSTANTS.C_MAX_MANIFOLDS DO
            VO_Manifold_Pumps[L_i] := FALSE;
        END_FOR;
    4:
        L_Target_Supply_Temp := LIMIT(GVL_CONSTANTS.C_BOILER_SETPOINT_MIN, L_Target_Supply_Temp - REAL#5.0, GVL_CONSTANTS.C_BOILER_SETPOINT_MAX);
    5:
        // Input-quality degradation is published for explainability first.
        // Runtime suppression remains governed by existing sensor validation
        // and safety/pressure ownership paths.
ELSE
    // no auto-recovery action
END_CASE;

fbValveTestManager(
    VI_System_Time_MS := VI_System_Time_MS,
    VI_IsActivePLC := VI_IsActivePLC,
    VI_Valve_Currents := VI_Manifold_Currents,
    VI_Valve_End_Switches := VI_Manifold_End_Switches,
    VI_Config := VI_Valve_Test_Config
);

IF fbValveTestManager.VO_Test_Active THEN
    L_i := fbValveTestManager.VO_Current_Valve;
    IF L_i >= 1 AND L_i <= GVL_CONSTANTS.C_MAX_MANIFOLDS THEN
        IF fbValveTestManager.VO_Valve_Cmd[L_i] THEN
            VO_Manifold_Valves[L_i] := REAL#100.0;
        ELSE
            VO_Manifold_Valves[L_i] := REAL#0.0;
        END_IF;
        VO_Manifold_Pumps[L_i] := FALSE;
    END_IF;
END_IF;

fbBoilerControl(
    VI_System_Time_MS := VI_System_Time_MS,
    VI_IsActivePLC := VI_IsActivePLC,
    VI_DHW_Heating_Demand := VI_DHW_Heating_Demand,
    VI_DHW_Target_Temp := VI_DHW_Target_Temp,
    VI_Target_Supply_Temp := L_Target_Supply_Temp,
    VI_Freeze_Mode_Active := L_Freeze_Active,
    VI_Policy_Degraded := L_Policy_Degraded,
    VI_Manifold_Pumps := VO_Manifold_Pumps,
    VI_Manifold_Valves := VO_Manifold_Valves,
    VI_Boiler_Flame_Status := VI_Boiler_Flame_Status,
    VI_Boiler_Error_Status := VI_Boiler_Error_Status,
    VI_Boiler_OT_Online := VI_Boiler_OT_Online,
    VI_Boiler_Modulation := VI_Boiler_Modulation,
    VO_Boiler_OT_Enable => VO_Boiler_OT_Enable,
    VO_Boiler_OT_Setpoint => VO_Boiler_OT_Setpoint,
    VO_Boiler_Status => VO_Boiler_Status,
    VO_Any_Subsystem_Degraded => L_Subsys_Degraded
);

GVL_STATE.G_Heating_Subsystem_Degraded := GVL_STATE.G_Heating_Subsystem_Degraded OR L_Subsys_Degraded;

// >>> BULK_SYNC_ANCHOR: FB_Heating_System_Manager <<<
          
END_FUNCTION_BLOCK

FUNCTION_BLOCK FB_Trend_Analyzer
  VAR_INPUT
    VI_Count : INT;
  END_VAR
  VAR_OUTPUT
    VO_Average : REAL;
    VO_Max : REAL;
    VO_Min : REAL;
    VO_Trend_Up : BOOL;
    VO_Trend_Down : BOOL;
  END_VAR
  VAR_IN_OUT
    VI_Data : ARRAY[1..GVL_CONSTANTS.C_MAX_TREND_DATA_POINTS] OF REAL;
  END_VAR
  VAR
    L_i : INT;
    L_Sum : REAL;
  END_VAR

            IF VI_Count > 0 AND VI_Count <= GVL_CONSTANTS.C_MAX_TREND_DATA_POINTS THEN
    VO_Max := VI_Data[1];
    VO_Min := VI_Data[1];
    L_Sum := 0.0;
    
    FOR L_i := 1 TO VI_Count DO
        IF VI_Data[L_i] > VO_Max THEN VO_Max := VI_Data[L_i]; END_IF;
        IF VI_Data[L_i] < VO_Min THEN VO_Min := VI_Data[L_i]; END_IF;
        L_Sum := L_Sum + VI_Data[L_i];
    END_FOR;
    
    VO_Average := L_Sum / INT_TO_REAL(VI_Count);
    
    IF VI_Count >= 2 THEN
        VO_Trend_Up := (VI_Data[VI_Count] > VI_Data[1]);
        VO_Trend_Down := (VI_Data[VI_Count] < VI_Data[1]);
    END_IF;
END_IF;
          
END_FUNCTION_BLOCK

FUNCTION_BLOCK FB_Water_Isolation_Runtime_Projection
  VAR_INPUT
    VI_Enable : BOOL;
    VI_System_Time_MS : UDINT;
  END_VAR
  VAR
    L_i : INT;
    L_Leak_State : ST_Water_Leak_Runtime_State;
    L_Isolation_State : ST_Water_Isolation_Runtime_State;
    L_Traversal : ST_Water_Graph_Traversal_State;
    L_Any_Isolation : BOOL;
    L_Any_Selective : BOOL;
    L_Global_Fallback : BOOL;
  END_VAR

            IF NOT VI_Enable THEN
    GVL_Water_Isolation_Runtime.G_Runtime_Valid := FALSE;
    RETURN;
END_IF;

FOR L_i := 1 TO GVL_CONSTANTS.C_MAX_FLOOD_SENSORS DO

    L_Leak_State := GVL_Water_Runtime_Projection.G_Leak_Runtime_State[L_i];
    L_Traversal := GVL_Water_Orchestration.G_Traversal_State[L_i];

    L_Isolation_State := (Projection_Valid := TRUE);
    L_Isolation_State.Projection_System_Time_MS := VI_System_Time_MS;

    L_Isolation_State.Hydraulic_Zone_Id := L_Leak_State.Hydraulic_Zone_Id;
    L_Isolation_State.Isolation_Group_Id := L_Leak_State.Isolation_Group_Id;
    L_Isolation_State.Valve_Group_Id := L_Traversal.Target_Valve_Group_Id;

    L_Isolation_State.Active_Global_Close_Path :=
        L_Leak_State.Active_Global_Close_Path;

    L_Isolation_State.Active_Safety_Latch :=
        L_Leak_State.Active_Safety_Leak_Latched;

    L_Isolation_State.Mapping_Valid :=
        L_Traversal.Traversal_Valid;

    L_Isolation_State.Fallback_To_Global_Required :=
        L_Traversal.Global_Fallback_Required;

    IF L_Leak_State.Leak_Confirmed THEN

        L_Isolation_State.Isolation_Requested := TRUE;

        IF L_Traversal.Selective_Path_Allowed
           AND NOT L_Traversal.Global_Fallback_Required THEN

            L_Isolation_State.Selective_Isolation_Requested := TRUE;
            L_Isolation_State.Reason_Code := 1;
            L_Isolation_State.Reason_Text :=
                'Selective orchestration path available';

        ELSE

            L_Isolation_State.Global_Isolation_Requested := TRUE;
            L_Isolation_State.Reason_Code := 2;
            L_Isolation_State.Reason_Text :=
                'Global fallback required';

        END_IF;

    END_IF;

    GVL_Water_Isolation_Runtime.G_Isolation_Runtime_State[L_i] :=
        L_Isolation_State;

    L_Any_Isolation :=
        L_Any_Isolation
        OR L_Isolation_State.Isolation_Requested;

    L_Any_Selective :=
        L_Any_Selective
        OR L_Isolation_State.Selective_Isolation_Requested;

    L_Global_Fallback :=
        L_Global_Fallback
        OR L_Isolation_State.Global_Isolation_Requested;

END_FOR;

GVL_Water_Isolation_Runtime.G_Any_Isolation_Requested :=
    L_Any_Isolation;

GVL_Water_Isolation_Runtime.G_Any_Selective_Isolation :=
    L_Any_Selective;

GVL_Water_Isolation_Runtime.G_Global_Fallback_Required :=
    L_Global_Fallback;

GVL_Water_Isolation_Runtime.G_Runtime_Valid := TRUE;
GVL_Water_Isolation_Runtime.G_Last_Update_MS := VI_System_Time_MS;

IF L_Global_Fallback THEN
    GVL_Water_Isolation_Runtime.G_Status_Code := 2;
    GVL_Water_Isolation_Runtime.G_Status_Text :=
        'Global isolation fallback required';
ELSIF L_Any_Selective THEN
    GVL_Water_Isolation_Runtime.G_Status_Code := 1;
    GVL_Water_Isolation_Runtime.G_Status_Text :=
        'Selective orchestration active';
ELSE
    GVL_Water_Isolation_Runtime.G_Status_Code := 0;
    GVL_Water_Isolation_Runtime.G_Status_Text :=
        'Isolation runtime active';
END_IF;
          
END_FUNCTION_BLOCK

FUNCTION_BLOCK FB_Heating_Runtime_Event_Manager
  VAR_INPUT
    VI_Enable : BOOL;
    VI_Event : ST_Heating_Runtime_Phase_Event;
  END_VAR
  VAR_OUTPUT
    VO_Event_Stored : BOOL;
    VO_Buffer_Overflow : BOOL;
    VO_Manager_Ready : BOOL;
    VO_Manager_Status_Code : UINT;
    VO_Manager_Status_Text : STRING(128);
  END_VAR
  VAR_IN_OUT
    VIO_Buffer : ST_Heating_Runtime_Event_Buffer;
  END_VAR
  VAR
    L_Write_Index : UINT;
  END_VAR

            // ==============================================================================
// Heating runtime event manager
// Read-only orchestration telemetry/event layer.
// DOES NOT own runtime.
// DOES NOT own heating logic.
// DOES NOT own diagnostics.
// DOES NOT own OpenTherm transport.
// ==============================================================================



// ======================================================
// DEFAULTS
// ======================================================
VO_Event_Stored := FALSE;
VO_Buffer_Overflow := FALSE;
VO_Manager_Ready := FALSE;
VO_Manager_Status_Code := 0;
VO_Manager_Status_Text := 'Heating runtime event manager disabled';

IF NOT VI_Enable THEN
    RETURN;
END_IF;

// ======================================================
// BUFFER VALIDATION
// ======================================================
IF VIO_Buffer.Write_Index > 32 THEN
    VIO_Buffer.Write_Index := 1;
END_IF;

IF VIO_Buffer.Read_Index > 32 THEN
    VIO_Buffer.Read_Index := 1;
END_IF;

// ======================================================
// WRITE INDEX
// ======================================================
L_Write_Index := VIO_Buffer.Write_Index + 1;

IF L_Write_Index > 32 THEN
    L_Write_Index := 1;
END_IF;

// ======================================================
// STORE EVENT
// ======================================================
VIO_Buffer.Events[L_Write_Index] := VI_Event;
VIO_Buffer.Write_Index := L_Write_Index;

IF VIO_Buffer.Event_Count < 32 THEN
    VIO_Buffer.Event_Count := VIO_Buffer.Event_Count + 1;
ELSE
    VIO_Buffer.Overflow := TRUE;
    VO_Buffer_Overflow := TRUE;
END_IF;

// ======================================================
// BUFFER INTEGRITY
// ======================================================
VIO_Buffer.Ordering_Integrity_Valid :=
    VI_Event.Ordering_Valid;

VIO_Buffer.Isolation_Integrity_Valid :=
    VI_Event.Isolation_Valid;

VIO_Buffer.Diagnostics_Visibility_Valid :=
    VI_Event.Diagnostics_Visible;

VIO_Buffer.Explainability_Visibility_Valid :=
    VI_Event.Explainability_Visible;

VIO_Buffer.OpenTherm_Ownership_Valid :=
    VI_Event.OpenTherm_Ownership_Valid;

VIO_Buffer.Cascade_Ownership_Valid :=
    VI_Event.Cascade_Ownership_Valid;

VIO_Buffer.Safety_Ownership_Valid :=
    VI_Event.Safety_Integrity_Valid;

VIO_Buffer.Lifecycle_Integrity_Valid :=
    NOT VI_Event.Event_Failed;

// ======================================================
// BUFFER STATUS
// ======================================================
IF VO_Buffer_Overflow THEN
    VIO_Buffer.Status_Code := 100;
    VIO_Buffer.Status_Text := 'Heating runtime event buffer overflow';
ELSE
    VIO_Buffer.Status_Code := 1;
    VIO_Buffer.Status_Text := 'Heating runtime event stored';
END_IF;

// ======================================================
// OUTPUT STATUS
// ======================================================
VO_Event_Stored := TRUE;
VO_Manager_Ready := TRUE;
VO_Manager_Status_Code := VIO_Buffer.Status_Code;
VO_Manager_Status_Text := VIO_Buffer.Status_Text;

// >>> BULK_SYNC_ANCHOR: FB_Heating_Runtime_Event_Manager <<<
          
END_FUNCTION_BLOCK

FUNCTION_BLOCK FB_Trend_Adapter
  VAR_INPUT
    VI_Data : ST_Trend_Data;
  END_VAR
  VAR_OUTPUT
    VO_Average : REAL;
    VO_Min : REAL;
    VO_Max : REAL;
    VO_Trend_Up : BOOL;
    VO_Trend_Down : BOOL;
  END_VAR
  VAR
    fbAnalyzer : FB_Trend_Analyzer;
    L_Data_Copy : ARRAY[1..GVL_CONSTANTS.C_MAX_TREND_DATA_POINTS] OF REAL;
    L_Count : INT;
    L_i : INT;
  END_VAR

            // Normalize count to analyzer bounds
L_Count := UDINT_TO_INT(VI_Data.record_count);
IF L_Count < 0 THEN
    L_Count := 0;
END_IF;
IF L_Count > GVL_CONSTANTS.C_MAX_TREND_DATA_POINTS THEN
    L_Count := GVL_CONSTANTS.C_MAX_TREND_DATA_POINTS;
END_IF;

// Copy source values into analyzer-compatible buffer
FOR L_i := 1 TO GVL_CONSTANTS.C_MAX_TREND_DATA_POINTS DO
    L_Data_Copy[L_i] := 0.0;
END_FOR;

IF L_Count > 0 THEN
    FOR L_i := 1 TO L_Count DO
        L_Data_Copy[L_i] := VI_Data.values[L_i];
    END_FOR;
END_IF;

fbAnalyzer(
    VI_Count := L_Count,
    VI_Data := L_Data_Copy,
    VO_Average => VO_Average,
    VO_Max => VO_Max,
    VO_Min => VO_Min,
    VO_Trend_Up => VO_Trend_Up,
    VO_Trend_Down => VO_Trend_Down
);
          
END_FUNCTION_BLOCK

FUNCTION_BLOCK FB_Water_Orchestration_Runtime
  VAR_INPUT
    VI_Enable : BOOL;
    VI_System_Time_MS : UDINT;
  END_VAR
  VAR
    L_i : INT;
    L_Path : ST_Water_Isolation_Path_Runtime_State;
    L_Traversal : ST_Water_Graph_Traversal_State;
    L_Orchestration : ST_Water_Orchestration_Runtime_State;
    L_Any_Conflict : BOOL;
    L_Any_Escalation : BOOL;
  END_VAR

            IF NOT VI_Enable THEN
    GVL_Water_Orchestration.G_Runtime_Valid := FALSE;
    RETURN;
END_IF;

FOR L_i := 1 TO GVL_CONSTANTS.C_MAX_FLOOD_SENSORS DO

    L_Path :=
        GVL_Water_Hydraulic_Graph.G_Isolation_Path[L_i];

    // Traversal runtime.
    L_Traversal := (Runtime_Valid := TRUE);

    L_Traversal.Runtime_System_Time_MS :=
        VI_System_Time_MS;

    L_Traversal.Sensor_Id := TO_UINT(L_i);

    L_Traversal.Start_Segment_Id :=
        L_Path.Active_Isolation_Group_Id;

    L_Traversal.Target_Valve_Group_Id :=
        L_Path.Active_Valve_Group_Id;

    L_Traversal.Shared_Trunk_Traversal :=
        L_Path.Shared_Trunk_Impact;

    L_Traversal.Upstream_Dependency_Detected :=
        L_Path.Shared_Trunk_Impact;

    L_Traversal.Downstream_Impact_Detected :=
        L_Path.Cross_Zone_Impact;

    L_Traversal.Traversal_Valid :=
        L_Path.Isolation_Path_Valid;

    L_Traversal.Traversal_Conflict :=
        L_Path.Conflict_Detected;

    L_Traversal.Traversal_Ambiguous :=
        L_Path.Isolation_Path_Ambiguous;

    IF L_Path.Multi_Valve_Path THEN
        L_Traversal.Dependency_Depth := 2;
    ELSE
        L_Traversal.Dependency_Depth := 1;
    END_IF;

    L_Traversal.Selective_Path_Allowed :=
        L_Path.Selective_Isolation_Allowed;

    L_Traversal.Global_Fallback_Required :=
        L_Path.Global_Fallback_Required;

    // Orchestration runtime.
    L_Orchestration := (Runtime_Valid := TRUE);

    L_Orchestration.Runtime_System_Time_MS :=
        VI_System_Time_MS;

    L_Orchestration.Isolation_Sequence_Active :=
        L_Traversal.Traversal_Valid;

    L_Orchestration.Shared_Trunk_Sequencing :=
        L_Traversal.Shared_Trunk_Traversal;

    L_Orchestration.Staged_Close_Required :=
        L_Path.Multi_Valve_Path;

    L_Orchestration.Recovery_Sequence_Active :=
        GVL_INTENT_SAFETY.I_Water_Selective_Recovery_Allowed;

    L_Orchestration.Staged_Open_Required :=
        L_Orchestration.Recovery_Sequence_Active
        AND L_Path.Multi_Valve_Path;

    L_Orchestration.Observation_Window_Active :=
        L_Orchestration.Recovery_Sequence_Active;

    // Conservative sequencing governance.
    IF L_Traversal.Traversal_Conflict
       OR L_Traversal.Traversal_Ambiguous THEN

        L_Orchestration.Rollback_Required := TRUE;
        L_Orchestration.Escalation_Required := TRUE;
        L_Orchestration.Sequencing_Valid := FALSE;

        L_Orchestration.Status_Code := 2;
        L_Orchestration.Status_Text :=
            'Orchestration conflict escalation active';

    ELSE

        L_Orchestration.Sequencing_Valid := TRUE;

        IF L_Orchestration.Shared_Trunk_Sequencing THEN
            L_Orchestration.Status_Code := 1;
            L_Orchestration.Status_Text :=
                'Shared trunk orchestration active';
        ELSE
            L_Orchestration.Status_Code := 0;
            L_Orchestration.Status_Text :=
                'Deterministic orchestration active';
        END_IF;

    END_IF;

    GVL_Water_Orchestration.G_Traversal_State[L_i] :=
        L_Traversal;

    GVL_Water_Orchestration.G_Orchestration_State[L_i] :=
        L_Orchestration;

    L_Any_Conflict :=
        L_Any_Conflict
        OR L_Traversal.Traversal_Conflict;

    L_Any_Escalation :=
        L_Any_Escalation
        OR L_Orchestration.Escalation_Required;

END_FOR;

GVL_Water_Orchestration.G_Topology_Version := 1;
GVL_Water_Orchestration.G_Config_Runtime_Ready := TRUE;

GVL_Water_Orchestration.G_Any_Traversal_Conflict :=
    L_Any_Conflict;

GVL_Water_Orchestration.G_Any_Escalation_Required :=
    L_Any_Escalation;

GVL_Water_Orchestration.G_Runtime_Valid := TRUE;
GVL_Water_Orchestration.G_Last_Update_MS := VI_System_Time_MS;

IF L_Any_Escalation THEN
    GVL_Water_Orchestration.G_Status_Code := 2;
    GVL_Water_Orchestration.G_Status_Text :=
        'Water orchestration escalation active';
ELSIF L_Any_Conflict THEN
    GVL_Water_Orchestration.G_Status_Code := 1;
    GVL_Water_Orchestration.G_Status_Text :=
        'Water orchestration conflict detected';
ELSE
    GVL_Water_Orchestration.G_Status_Code := 0;
    GVL_Water_Orchestration.G_Status_Text :=
        'Water orchestration runtime healthy';
END_IF;
          
END_FUNCTION_BLOCK

FUNCTION_BLOCK FB_Ventilation_System_Manager
  VAR_INPUT
    VI_System_Time_MS : UDINT;
    VI_IsActivePLC : BOOL;
    VI_Outdoor_Temp : REAL;
    VI_Current_Scenario : E_SCENARIO_TYPE;
    VI_System_Mode : E_System_Operating_Mode;
    VI_Config : ST_Ventilation_Global_Config;
    VI_Fire_Alarm : BOOL;
    VI_Gas_Alarm : BOOL;
    VI_PV3_Boost_Req : BOOL;
    VI_Supply_100_Req : BOOL;
    VI_Exhaust_100_Req : BOOL;
    VI_Supply_80_Req : BOOL;
    VI_Vent_Stop : BOOL;
    VI_IO_Modules_Online : ARRAY[1..GVL_CONSTANTS.C_MAX_MODULES] OF BOOL;
  END_VAR
  VAR_OUTPUT
    VO_Supply_Fans : ARRAY[1..GVL_CONSTANTS.C_MAX_SUPPLY_FANS] OF BYTE;
    VO_Exhaust_Fans : ARRAY[1..GVL_CONSTANTS.C_MAX_EXHAUST_FANS] OF BYTE;
    VO_Heater_Power : ARRAY[1..GVL_CONSTANTS.C_MAX_BOILERS] OF REAL;
    VO_Status_Msg : STRING(200);
    VO_Ventilation_IO_Fault : BOOL;
    VO_Ventilation_Subsystem_Degraded : BOOL;
  END_VAR
  VAR_IN_OUT
    VI_Supply_Temps : ARRAY[1..GVL_CONSTANTS.C_MAX_SUPPLY_TEMPS] OF REAL;
    VI_Room_Temps : ARRAY[1..16] OF REAL;
    VI_Room_Humidities : ARRAY[1..16] OF REAL;
    VI_Room_CO2 : ARRAY[1..16] OF REAL;
    VI_Wet_Zone_Active : ARRAY[1..GVL_CONSTANTS.C_MAX_WET_ZONES] OF BOOL;
    VI_Rule_Actions : ARRAY[1..GVL_CONSTANTS.C_MAX_RULES] OF ST_Rule_Action;
  END_VAR
  VAR
    L_Policy_Normal : BOOL;
    L_Policy_Safe_Stop : BOOL;
    L_Policy_Degraded : BOOL;
    L_Policy_Freeze_Protection : BOOL;
    L_i : INT;
    L_j : INT;
    L_Max_CO2 : REAL;
    L_Max_Hum : REAL;
    L_Base_Speed : BYTE;
    L_Target_Temp : REAL;
    L_PID_Heaters : ARRAY[1..GVL_CONSTANTS.C_MAX_BOILERS] OF FB_PID_Controller;
    L_Wet_Zone_Timers : ARRAY[1..GVL_CONSTANTS.C_MAX_WET_ZONES] OF FB_System_Timer_TOF;
  END_VAR

            // ========================================
// Ventilation policy layer
// ========================================
VO_Ventilation_IO_Fault := FALSE;
VO_Ventilation_Subsystem_Degraded := FALSE;
L_Policy_Normal := (VI_System_Mode = E_System_Operating_Mode.MODE_NORMAL);
L_Policy_Safe_Stop := (VI_System_Mode = E_System_Operating_Mode.MODE_SAFE_STOP);
L_Policy_Degraded := (VI_System_Mode = E_System_Operating_Mode.MODE_DEGRADED);
L_Policy_Freeze_Protection := (VI_System_Mode = E_System_Operating_Mode.MODE_FREEZE_PROTECTION);

IF NOT VI_IsActivePLC THEN
    FOR L_i := 1 TO GVL_CONSTANTS.C_MAX_SUPPLY_FANS DO
        VO_Supply_Fans[L_i] := 0;
        IF L_i <= GVL_CONSTANTS.C_MAX_SUPPLY_TEMPS THEN
            VO_Heater_Power[L_i] := 0.0;
        END_IF;
    END_FOR;
    FOR L_i := 1 TO GVL_CONSTANTS.C_MAX_EXHAUST_FANS DO
        VO_Exhaust_Fans[L_i] := 0;
    END_FOR;
    VO_Status_Msg := 'ВЕНТИЛЯЦИЯ: РЕЗЕРВНЫЙ ПЛК';
    RETURN;
END_IF;

// Проверка связи с модулями ввода-вывода
FOR L_i := 1 TO GVL_CONSTANTS.C_MAX_MODULES DO
    IF NOT VI_IO_Modules_Online[L_i] THEN
        VO_Ventilation_IO_Fault := TRUE;
        FOR L_j := 1 TO GVL_CONSTANTS.C_MAX_SUPPLY_FANS DO
            VO_Supply_Fans[L_j] := 0;
        END_FOR;
        FOR L_j := 1 TO GVL_CONSTANTS.C_MAX_EXHAUST_FANS DO
            VO_Exhaust_Fans[L_j] := 0;
        END_FOR;
        FOR L_j := 1 TO GVL_CONSTANTS.C_MAX_BOILERS DO
            VO_Heater_Power[L_j] := 0.0;
        END_FOR;
        VO_Status_Msg := 'ОШИБКА: Потеря связи с модулями ввода-вывода';
        RETURN;
    END_IF;
END_FOR;

// =========================
// SYSTEM MODE / HARD REQUEST OVERRIDES
// =========================
IF L_Policy_Safe_Stop OR VI_Vent_Stop THEN
    FOR L_i := 1 TO GVL_CONSTANTS.C_MAX_SUPPLY_FANS DO
        VO_Supply_Fans[L_i] := 0;
    END_FOR;
    FOR L_i := 1 TO GVL_CONSTANTS.C_MAX_EXHAUST_FANS DO
        VO_Exhaust_Fans[L_i] := 0;
    END_FOR;
    FOR L_i := 1 TO GVL_CONSTANTS.C_MAX_BOILERS DO
        VO_Heater_Power[L_i] := 0.0;
    END_FOR;
    IF VI_Vent_Stop THEN
        VO_Status_Msg := 'ВЕНТИЛЯЦИЯ: ОСТАНОВЛЕНА ПО КОМАНДЕ';
    ELSE
        VO_Status_Msg := 'ВЕНТИЛЯЦИЯ: ОСТАНОВЛЕНА POLICY SAFE_STOP';
    END_IF;
    RETURN;
END_IF;

IF L_Policy_Degraded THEN
    FOR L_i := 1 TO GVL_CONSTANTS.C_MAX_SUPPLY_FANS DO
        VO_Supply_Fans[L_i] := 0;
    END_FOR;
    FOR L_i := 1 TO GVL_CONSTANTS.C_MAX_BOILERS DO
        VO_Heater_Power[L_i] := 0.0;
    END_FOR;
    VO_Ventilation_Subsystem_Degraded := TRUE;
    VO_Status_Msg := 'ВЕНТИЛЯЦИЯ: DEGRADED POLICY';
END_IF;

IF L_Policy_Freeze_Protection THEN
    FOR L_i := 1 TO GVL_CONSTANTS.C_MAX_SUPPLY_FANS DO
        VO_Supply_Fans[L_i] := 0;
    END_FOR;
    FOR L_i := 1 TO GVL_CONSTANTS.C_MAX_EXHAUST_FANS DO
        VO_Exhaust_Fans[L_i] := 0;
    END_FOR;
    FOR L_i := 1 TO GVL_CONSTANTS.C_MAX_BOILERS DO
        VO_Heater_Power[L_i] := 0.0;
    END_FOR;
    VO_Status_Msg := 'ВЕНТИЛЯЦИЯ: FREEZE_PROTECTION POLICY (stop)';
    RETURN;
END_IF;

// 1. Определение базовой скорости и целевой температуры по сценарию (ТЗ 7.1)
CASE VI_Current_Scenario OF
    E_SCENARIO_TYPE.SCENARIO_AWAY:
        L_Base_Speed := VI_Config.Scenario_Modes[3].Base_Fan_Speed;
        L_Target_Temp := VI_Config.Scenario_Modes[3].Target_Temp;
    E_SCENARIO_TYPE.SCENARIO_SLEEP:
        L_Base_Speed := VI_Config.Scenario_Modes[2].Base_Fan_Speed;
        L_Target_Temp := VI_Config.Scenario_Modes[2].Target_Temp;
    ELSE // PRESENCE, MORNING, EVENING
        L_Base_Speed := VI_Config.Scenario_Modes[1].Base_Fan_Speed;
        L_Target_Temp := VI_Config.Scenario_Modes[1].Target_Temp;
END_CASE;

// 2. Логика управления приточными установками (П-1, П-2, П-3)
FOR L_i := 1 TO GVL_CONSTANTS.C_MAX_SUPPLY_FANS DO
    IF L_i <= GVL_CONSTANTS.C_MAX_SUPPLY_TEMPS THEN
        L_PID_Heaters[L_i](
            VI_SetPoint := L_Target_Temp,
            VI_ProcessValue := VI_Supply_Temps[L_i],
            VI_Kp := 4.0, VI_Tn := 120.0, VI_Tv := 0.0,
            VI_Y_Min := 0.0, VI_Y_Max := 100.0, VI_Cycle_Time_S := 1.0,
            VO_Output => VO_Heater_Power[L_i]
        );
    END_IF;

    VO_Supply_Fans[L_i] := L_Base_Speed;

    FOR L_j := 1 TO GVL_CONSTANTS.C_MAX_RULES DO
        IF VI_Rule_Actions[L_j].Active AND VI_Rule_Actions[L_j].Target_ID = L_i THEN
            IF VI_Rule_Actions[L_j].Action_Type = E_Rule_Action_Type.ACTION_SET_VENTILATION THEN
                VO_Supply_Fans[L_i] := REAL_TO_BYTE(VI_Rule_Actions[L_j].Value);
            END_IF;
        END_IF;
    END_FOR;
END_FOR;

// 3. Логика управления вытяжными установками (В-1 .. В-5)
FOR L_i := 1 TO GVL_CONSTANTS.C_MAX_EXHAUST_FANS DO
    VO_Exhaust_Fans[L_i] := L_Base_Speed;

    FOR L_j := 1 TO GVL_CONSTANTS.C_MAX_WET_ZONES DO
        IF VI_Config.wet_zone_to_exhaust_map[L_j] = L_i THEN
            L_Wet_Zone_Timers[L_j](IN := VI_Wet_Zone_Active[L_j], PT := T#5m, VI_System_Time_MS := VI_System_Time_MS);
            IF VI_Wet_Zone_Active[L_j] THEN
                VO_Exhaust_Fans[L_i] := 80;
            ELSIF L_Wet_Zone_Timers[L_j].Q THEN
                VO_Exhaust_Fans[L_i] := 50;
            END_IF;
        END_IF;
    END_FOR;
END_FOR;

// ========================================
// OPERATIONAL REQUEST OVERRIDES
// ========================================
IF VI_Supply_100_Req THEN
    FOR L_i := 1 TO GVL_CONSTANTS.C_MAX_SUPPLY_FANS DO
        VO_Supply_Fans[L_i] := 100;
    END_FOR;
ELSIF VI_Supply_80_Req THEN
    FOR L_i := 1 TO GVL_CONSTANTS.C_MAX_SUPPLY_FANS DO
        IF VO_Supply_Fans[L_i] < 80 THEN
            VO_Supply_Fans[L_i] := 80;
        END_IF;
    END_FOR;
END_IF;

IF VI_PV3_Boost_Req THEN
    IF GVL_CONSTANTS.C_MAX_SUPPLY_FANS >= 3 THEN
        VO_Supply_Fans[3] := 100;
    END_IF;
END_IF;

IF VI_Exhaust_100_Req THEN
    FOR L_i := 1 TO GVL_CONSTANTS.C_MAX_EXHAUST_FANS DO
        VO_Exhaust_Fans[L_i] := 100;
    END_FOR;
END_IF;

// ========================================
// VENT_FINAL_CLAMP
// ========================================
IF L_Policy_Degraded THEN
    FOR L_i := 1 TO GVL_CONSTANTS.C_MAX_EXHAUST_FANS DO
        VO_Exhaust_Fans[L_i] := MIN(VO_Exhaust_Fans[L_i], VI_Config.Degraded_Exhaust_Limit);
    END_FOR;
END_IF;

// 4. Формирование статусного сообщения
IF L_Policy_Degraded THEN
    VO_Status_Msg := 'ВЕНТИЛЯЦИЯ: DEGRADED POLICY';
ELSIF VI_PV3_Boost_Req OR VI_Supply_100_Req OR VI_Exhaust_100_Req OR VI_Supply_80_Req THEN
    VO_Status_Msg := 'Вентиляция: активен операционный boost/request';
ELSE
    VO_Status_Msg := 'Вентиляция работает в штатном режиме';
END_IF;
// >>> BULK_SYNC_ANCHOR: FB_Ventilation_System_Manager <<<
          
END_FUNCTION_BLOCK

FUNCTION_BLOCK FB_Boiler_OpenTherm_Interface
  VAR_INPUT
    VI_Enable : ARRAY[1..GVL_CONSTANTS.C_MAX_BOILERS] OF BOOL;
    VI_Setpoint : ARRAY[1..GVL_CONSTANTS.C_MAX_BOILERS] OF REAL;
    VI_OT_Online : ARRAY[1..GVL_CONSTANTS.C_MAX_BOILERS] OF BOOL;
    VI_OT_Error : ARRAY[1..GVL_CONSTANTS.C_MAX_BOILERS] OF BOOL;
  END_VAR
  VAR_OUTPUT
    VO_OT_Enable : ARRAY[1..GVL_CONSTANTS.C_MAX_BOILERS] OF BOOL;
    VO_OT_Setpoint : ARRAY[1..GVL_CONSTANTS.C_MAX_BOILERS] OF REAL;
    VO_OT_Command_Valid : ARRAY[1..GVL_CONSTANTS.C_MAX_BOILERS] OF BOOL;
  END_VAR
  VAR
    L_i : INT;
    L_Setpoint : REAL;
    L_Setpoint_x10 : UINT;
    L_Command_Enable : BOOL;
    L_Command_Changed : BOOL;
    L_Last_Command_Enable : ARRAY[1..GVL_CONSTANTS.C_MAX_BOILERS] OF BOOL;
    L_Last_Command_Setpoint_x10 : ARRAY[1..GVL_CONSTANTS.C_MAX_BOILERS] OF UINT;
  END_VAR

            FOR L_i := 1 TO GVL_CONSTANTS.C_MAX_BOILERS DO

    VO_OT_Enable[L_i] := FALSE;
    VO_OT_Setpoint[L_i] := 0.0;
    VO_OT_Command_Valid[L_i] := FALSE;

    L_Command_Enable := FALSE;
    L_Setpoint := 0.0;
    L_Setpoint_x10 := 0;

    // ======================================================
    // COMMAND VALIDATION
    // ======================================================
    IF VI_Enable[L_i] AND VI_OT_Online[L_i] AND NOT VI_OT_Error[L_i] THEN
        L_Command_Enable := TRUE;
        L_Setpoint := LIMIT(20.0, VI_Setpoint[L_i], 80.0);
        L_Setpoint_x10 := REAL_TO_UINT(L_Setpoint * 10.0);

        VO_OT_Enable[L_i] := TRUE;
        VO_OT_Setpoint[L_i] := L_Setpoint;
    END_IF;

    // ======================================================
    // PHYSICAL ADAPTER COMMAND IMAGE
    // ======================================================
    GVL_OPENTHERM_ADAPTER.G_Command[L_i].Enable := L_Command_Enable;
    GVL_OPENTHERM_ADAPTER.G_Command[L_i].Setpoint_x10 := L_Setpoint_x10;

